			// Set ACK Timestamp	
			_TmpAlarm.AckDateTime[0] := TO_DINT(_TempTimestruct.wYear);
			_TmpAlarm.AckDateTime[1] := TO_DINT(_TempTimestruct.wMonth);
			_TmpAlarm.AckDateTime[2] := TO_DINT(_TempTimestruct.wDay);
			_TmpAlarm.AckDateTime[3] := TO_DINT(_TempTimestruct.wHour);
			_TmpAlarm.AckDateTime[4] := TO_DINT(_TempTimestruct.wMinute);
			_TmpAlarm.AckDateTime[5] := TO_DINT(_TempTimestruct.wSecond);
			_TmpAlarm.AckDateTime[6] := TO_DINT(_TempTimestruct.wMilliseconds);
			_TmpAlarm.Trigger		 := FALSE;

			// Move to History	
			_hr := THIS^.AlarmArrayHandler(NewAlarm_Ref			:= _TmpAlarm,
										   ActAlarmsCounter_Ref := THIS^.MsgInHistory,
										   MaxArrayElements		:= Tc3_PackML_V2.MaxHistoryAlarms,
										   pAlarmArray			:= ADR(_AdminTag.AlarmHistory),
										   BufferOverflow_Ref	:= _BufferOverflow);

			IF _BufferOverflow THEN
				Tc2_System.ADSLOGSTR(msgCtrlMask := Tc2_System.ADSLOG_MSGTYPE_ERROR, msgFmtStr := Tc2_Standard.CONCAT(cBaseMsg, 'MoveAlarmToHistory: %s'), strArg := 'History Buffer is full / FIFO active');
			END_IF

			IF Tc3_Module.SUCCEEDED(_hr) THEN
				// Close empty entry in source array
				Tc2_System.MEMMOVE(destAddr := ADR(pAlarmArray[_Iterator]), srcAddr := ADR(pAlarmArray[_Iterator + 1]), n := (SIZEOF(Tc3_PackML_V2.ST_Alarm) * (TO_UINT((_MaxArrayElementsInternal) - (_Iterator))))); // move Alarm 
				Tc2_System.MEMSET(destAddr := ADR(pAlarmArray[_MaxArrayElementsInternal]), fillByte := 0, n := SIZEOF(Tc3_PackML_V2.ST_Alarm));																		   // delete last entry

				// Find next empty entry index 
				FOR _Iterator2 := 0 TO (_MaxArrayElementsInternal) DO
					IF (pAlarmArray[_Iterator2].Message = '') OR (_Iterator2 = _MaxArrayElementsInternal) THEN
						IF _Iterator2 > 0 THEN
							ActAlarms_Ref := _Iterator2 - 1;
						ELSE
							ActAlarms_Ref := _Iterator2;
						END_IF

						EXIT;
					END_IF
				END_FOR
			END_IF

			EXIT;
		END_IF
	END_FOR

	MoveAlarmToHistory := S_OK;
ELSE
	// Set internal Error
	Tc2_System.ADSLOGSTR(msgCtrlMask := cMsgCtrlMask, msgFmtStr := Tc2_Standard.CONCAT(cBaseMsg, 'MoveAlarmToHistory: %s'), strArg := 'Input-reference error');
	MoveAlarmToHistory := E_FAIL;
	_InternalError	   := TRUE;
END_IF
END_METHOD

PROPERTY Name : STRING
GET
END_GET
SET
_Name := Name;
END_SET
END_PROPERTY

METHOD OnAlarmCleared : HRESULT
VAR_INPUT
	fbEvent : REFERENCE TO FB_TcEvent; // Reference to FB_Event (Callback!)
END_VAR

VAR_INST
	_idxEventReceived : INT; // Event index
END_VAR

VAR
	_hr : HRESULT; // hresult
END_VAR
// Move Alarm to History
IF fbEvent.eSeverity = TcEventSeverity.Critical THEN // Check "Critical" --> Stop reason
	_hr := MoveAlarmToHistory(MaxArrayElements := Tc3_PackML_V2.MaxStopReasons,
							  EventId		   := fbEvent.nEventId,
							  pAlarmArray	   := ADR(_AdminTag.StopReason),
							  Timestamp		   := fbEvent.nTimestamp,
							  ActAlarms_Ref	   := UnclearedStopReasons);
ELSIF fbEvent.eSeverity = TcEventSeverity.Error THEN // Check "Error" --> Alarm
	_hr := MoveAlarmToHistory(MaxArrayElements := Tc3_PackML_V2.MaxAlarms,
							  EventId		   := fbEvent.nEventId,
							  pAlarmArray	   := ADR(_AdminTag.Alarm),
							  Timestamp		   := fbEvent.nTimestamp,
							  ActAlarms_Ref	   := UnclearedAlarms);

	IF _AlarmToStopReason AND Tc3_Module.SUCCEEDED(_hr) THEN
		_hr := THIS^.ClearStopReason(pAlarmArray	  := ADR(_AdminTag.StopReason),
									 ActAlarms_Ref	  := THIS^.UnclearedStopReasons,
									 MaxArrayElements := Tc3_PackML_V2.MaxStopReasons,
									 EventId		  := fbEvent.nEventId);
	END_IF
ELSIF fbEvent.eSeverity = TcEventSeverity.Warning THEN // Check "Warning" --> Warning
	_hr := MoveAlarmToHistory(MaxArrayElements := Tc3_PackML_V2.MaxWarnings,
							  EventId		   := fbEvent.nEventId,
							  pAlarmArray	   := ADR(_AdminTag.Warning),
							  Timestamp		   := fbEvent.nTimestamp,
							  ActAlarms_Ref	   := UnclearedWarnings);

	IF _WarningToStopReason AND Tc3_Module.SUCCEEDED(_hr) THEN
		_hr := THIS^.ClearStopReason(pAlarmArray	  := ADR(_AdminTag.StopReason),
									 ActAlarms_Ref	  := THIS^.UnclearedStopReasons,
									 MaxArrayElements := Tc3_PackML_V2.MaxStopReasons,
									 EventId		  := fbEvent.nEventId);
	END_IF
END_IF

OnAlarmCleared := S_OK; // in order to receive more callbacks (Set <> S_OK in order to cancel the callbacks for this program cycle.)
END_METHOD

// Callback Method
METHOD OnAlarmConfirmed : HRESULT
VAR_INPUT
	fbEvent : REFERENCE TO FB_TcEvent; // Reference to FB_Event (Callback!)
END_VAR

VAR
	_hr : HRESULT; // hresult
END_VAR
// Move Alarm to History
IF __ISVALIDREF(fbEvent) THEN
	// Set ACK Timestamp
	IF fbEvent.eSeverity = TcEventSeverity.Critical THEN // Check "Critical" --> Stop reason
		_hr := ConfirmAlarm(MaxArrayElements := Tc3_PackML_V2.MaxStopReasons,
							EventId			 := fbEvent.nEventId,
							pAlarmArray		 := ADR(_AdminTag.StopReason),
							Timestamp		 := fbEvent.nTimestamp,
							ActAlarms_Ref	 := UnclearedStopReasons);
	ELSIF fbEvent.eSeverity = TcEventSeverity.Error THEN // Check "Error" --> Alarm
		_hr := ConfirmAlarm(MaxArrayElements := Tc3_PackML_V2.MaxAlarms,
							EventId			 := fbEvent.nEventId,
							pAlarmArray		 := ADR(_AdminTag.Alarm),
							Timestamp		 := fbEvent.nTimestamp,
							ActAlarms_Ref	 := UnclearedAlarms);
	ELSIF fbEvent.eSeverity = TcEventSeverity.Warning THEN // Check "Warning" --> Warning
		_hr := ConfirmAlarm(MaxArrayElements := Tc3_PackML_V2.MaxWarnings,
							EventId			 := fbEvent.nEventId,
							pAlarmArray		 := ADR(_AdminTag.Warning),
							Timestamp		 := fbEvent.nTimestamp,
							ActAlarms_Ref	 := UnclearedWarnings);
	END_IF

	OnAlarmConfirmed := S_OK; // in order to receive more callbacks (Set <> S_OK in order to cancel the callbacks for this program cycle.)
ELSE
	// Set internal Error
	Tc2_System.ADSLOGSTR(msgCtrlMask := cMsgCtrlMask, msgFmtStr := Tc2_Standard.CONCAT(cBaseMsg, 'OnAlarmConfirmed: %s'), strArg := 'Input-reference error');
	OnAlarmConfirmed := E_FAIL;
	_InternalError	 := TRUE;
END_IF
END_METHOD

// Callback Method
METHOD OnAlarmRaised : HRESULT
VAR_INPUT
	fbEvent : REFERENCE TO FB_TcEvent; // Reference to FB_Event (Callback!)
END_VAR

VAR
	_TempTimestruct : TIMESTRUCT; // TimeStruct for ACK Time
END_VAR
// when (new) event is triggered -> trigger within cyclic method 'execute'
THIS^.NewEvent := TRUE;

//for local event -> raise counter
CntAlarmsRaised := CntAlarmsRaised + 1;

// save eventinfo locally
THIS^.stEventInfo.Source	  := fbEvent.ipSourceInfo.sName;
THIS^.stEventInfo.eSeverity	  := fbEvent.eSeverity;
THIS^.stEventInfo.EventClass  := fbEvent.EventClass;
THIS^.stEventInfo.EventId	  := fbEvent.nEventId;
THIS^.stEventInfo.ipArguments := fbEvent.ipArguments;

// TimeZone
fbSpecificLocalTime(in := Tc2_Utilities.FILETIME64_TO_SYSTEMTIME(fbEvent.nTimestamp), tzInfo := fbTimeZone.tzInfo, out => _TempTimestruct);

// Timestamp	
THIS^.stEventInfo.TimeRaised[0] := TO_DINT(_TempTimestruct.wYear);
THIS^.stEventInfo.TimeRaised[1] := TO_DINT(_TempTimestruct.wMonth);
THIS^.stEventInfo.TimeRaised[2] := TO_DINT(_TempTimestruct.wDay);
THIS^.stEventInfo.TimeRaised[3] := TO_DINT(_TempTimestruct.wHour);
THIS^.stEventInfo.TimeRaised[4] := TO_DINT(_TempTimestruct.wMinute);
THIS^.stEventInfo.TimeRaised[5] := TO_DINT(_TempTimestruct.wSecond);
THIS^.stEventInfo.TimeRaised[6] := TO_DINT(_TempTimestruct.wMilliseconds);
Tc2_System.MEMSET(destAddr := ADR(stEventInfo.TimeCleared), fillByte := 0, n := SIZEOF(stEventInfo.TimeCleared));
Tc2_System.MEMSET(destAddr := ADR(stEventInfo.TimeConfirmed), fillByte := 0, n := SIZEOF(stEventInfo.TimeConfirmed));

//store event info globally
aEventInfoBuffer[CntAlarmsRaised] := stEventInfo;

// activate requests in event triggered method 'OnMessageSent' to get related request info
aEventInfoBuffer[CntAlarmsRaised].fbRequestEventText.Request(eventClass := aEventInfoBuffer[CntAlarmsRaised].EventClass,
															 nEventId	:= aEventInfoBuffer[CntAlarmsRaised].EventId,
															 nLangId	:= 1033,
															 ipArgs		:= aEventInfoBuffer[CntAlarmsRaised].ipArguments);

OnAlarmRaised := S_OK; // in order to receive more callbacks (Set <> S_OK in order to cancel the callbacks for this program cycle.)
END_METHOD

PROPERTY ParentResponseDefinitions : ARRAY[0..4] OF SPT_BaseTypes.E_AlarmResponse
GET
ParentResponseDefinitions := _ParentResponseDefinitions;
END_GET
SET
_ParentResponseDefinitions := ParentResponseDefinitions;
END_SET
END_PROPERTY

METHOD Reset : BOOL
//This may or may not be called depending on the component type 

//which derives FB_ComponentBase
F_ClearAllEventsInClass(PackMLEventHandlerAlarms);
Reset := TRUE;
END_METHOD

METHOD PUBLIC TimeZone : BOOL
VAR_INST
	_Step : USINT; // Step Variable
END_VAR
CASE _Step OF
	0: // Start to get local Timezone 
		fbTimeZone.bExecute := TRUE;
		IF fbTimeZone.bBusy THEN
			_Step := _Step + 1;
		END_IF

	1: // set 
		fbTimeZone.bExecute := FALSE;
		_Step				:= 0;
		TimeZone			:= TRUE;

ELSE
	Tc2_System.ADSLOGSTR(msgCtrlMask := cMsgCtrlMask, msgFmtStr := Tc2_Standard.CONCAT(cBaseMsg, 'TimeZone: %s'), strArg := 'Case Idx error');
	_InternalError := TRUE;
END_CASE

fbTimeZone(sNetID := '');
IF fbTimeZone.bError THEN
	Tc2_System.ADSLOGSTR(msgCtrlMask := cMsgCtrlMask, msgFmtStr := Tc2_Standard.CONCAT(cBaseMsg, 'fbTimeZone ErrID: %s'), strArg := TO_STRING(fbTimeZone.nErrID));
	_InternalError := TRUE;
END_IF
END_METHOD

PROPERTY WarningToStopReason : BOOL
SET
_WarningToStopReason := WarningToStopReason;
END_SET
END_PROPERTY

METHOD PRIVATE WriteAlarmTags : HRESULT;
VAR_INPUT
	Alarm_Ref	  : REFERENCE TO Tc3_PackML_V2.ST_Alarm; // Reference to ST_Alarm of an new Alarm / Warning / Stop reason
	EventInfo_Ref : REFERENCE TO ST_EventInfo;			 // Reference to ST_EventInfo
	Trigger		  : BOOL;								 // Set / Reset Trigger in PML Structure
	AlarmIndex	  : DINT;								 // Alarm index
END_VAR
IF __ISVALIDREF(Alarm_Ref) AND __ISVALIDREF(EventInfo_Ref) THEN
	Alarm_Ref.ID	   := TO_DINT(EventInfo_Ref.EventId);
	Alarm_Ref.Value	   := AlarmIndex;
	Alarm_Ref.Message  := EventInfo_Ref.EventText;
	Alarm_Ref.Category := TO_DINT(EventInfo_Ref.eSeverity); // Verbose:=0, Info:=1, Warning:=2, Error:=3, Critical:=4
	Alarm_Ref.Trigger  := Trigger;
	Alarm_Ref.DateTime := EventInfo_Ref.TimeRaised;
	WriteAlarmTags	   := S_OK;
ELSE
	// Set internal Error
	Tc2_System.ADSLOGSTR(msgCtrlMask := cMsgCtrlMask, msgFmtStr := Tc2_Standard.CONCAT(cBaseMsg, 'WriteAlarmTags: %s'), strArg := 'Input-reference error');
	WriteAlarmTags := E_FAIL;
	_InternalError := TRUE;
END_IF
END_METHOD

END_FUNCTION_BLOCK

// Project Information/F_GetCompany
// This function has been automatically generated from the project information.
{attribute 'signature_flag' := '1073741824'}
{attribute 'TcGenerated'}
{attribute 'no-analysis'}
FUNCTION F_GetCompany : WSTRING
VAR_INPUT
	
END_VAR

F_GetCompany := "Beckhoff Automation LLC";

END_FUNCTION

// Project Information/F_GetTitle
// This function has been automatically generated from the project information.
{attribute 'signature_flag' := '1073741824'}
{attribute 'TcGenerated'}
{attribute 'no-analysis'}
FUNCTION F_GetTitle : WSTRING
VAR_INPUT
	
END_VAR

F_GetTitle := "SPT Components";

END_FUNCTION

// Project Information/F_GetVersion
// This function has been automatically generated from the project information.
{attribute 'signature_flag' := '1073741824'}
{attribute 'TcGenerated'}
{attribute 'no-analysis'}
FUNCTION F_GetVersion : ST_LibVersion
VAR_INPUT
	
END_VAR

F_GetVersion.iMajor := 3;
F_GetVersion.iMinor := 2;
F_GetVersion.iBuild := 6;
F_GetVersion.iRevision := 0;
F_GetVersion.sVersion := '3.2.6';
F_GetVersion.nFlags := 1;

END_FUNCTION

// Sensors/FB_DigitalSensor
FUNCTION_BLOCK FB_DigitalSensor EXTENDS FB_ComponentBase IMPLEMENTS I_DigitalSensorBase
VAR
	HardwareInput AT %I*		: BOOL;			  //Hardware input bit from the hysical sensor
	_DebounceMode				: E_DebounceMode; //Defines the debounce model that will filter the sensor's output to the program
	_DebounceTime				: TIME;			  //Time input parameter for use in Debounce functionality
	_Inverted					: BOOL;			  //Defines the output polarity of the sensor - a "TRUE" value will result in the signal of the sensor being inverted
	_SimulationInput			: BOOL;			  //Provides configuration input to the simulation functionality
	_SimulationTimebase			: UDINT;
	_SimulationMode				: E_SensorSimulationMode; //Defines the mode of operation for the simulation functionality of this component
	_TimeActive					: TIME;					  //Tracks the amount of time that the sensor has been in an active state
	_TimeInactive				: TIME;					  //Tracks the amount of time that the sensor has been in an inactive state
	_Active						: BOOL;
	TON_ActiveTimer				: Tc2_Standard.TON; //Tracks the amount of time that the sensor has been in an active state
	TON_InactiveTimer			: Tc2_Standard.TON; //Tracks the amount of time that the sensor has been in an inactive state
	TON_DebounceTimer			: Tc2_Standard.TON; //Utilized in the debounce implementation
	TP_DebounceTimer			: Tc2_Standard.TP;	//Utilized in the debounce implementation
	DigitalSensor_HMI			: ST_DigitalSensor_HMI;
	SimulationPulse1_TP			: Tc2_Standard.TP; //Pulse Timer for simulated sensor pulse generation
	SimulationPulse2_TP			: Tc2_Standard.TP; //Pulse Timer for simulated sensor pulse generation
	HMICommand_DigitalSensor_RT : R_TRIG;
END_VAR

METHOD PUBLIC CyclicLogic
VAR_INPUT
END_VAR
SUPER^.CyclicLogic();
IF _Simulate THEN
	CASE _SimulationMode OF
		E_SensorSimulationMode.InputDriven:
			_Active := _SimulationInput;

		E_SensorSimulationMode.Periodic:
			SimulationPulse1_TP(IN := NOT SimulationPulse2_TP.Q, PT := UDINT_TO_TIME(_SimulationTimebase));
			SimulationPulse2_TP(IN := NOT SimulationPulse1_TP.Q, PT := UDINT_TO_TIME(_SimulationTimebase));
			_Active := SimulationPulse2_TP.Q;
	END_CASE
ELSE
	_Active := ProcessInput(Input := HardwareInput);
END_IF
END_METHOD

PROPERTY Active : BOOL
GET
Active := _Active;
END_GET
END_PROPERTY

PROPERTY DebounceMode : E_DebounceMode
GET
DebounceMode := _DebounceMode;
END_GET
SET
_DebounceMode := DebounceMode;
END_SET
END_PROPERTY

PROPERTY DebounceTime : TIME
GET
DebounceTime := _DebounceTime;
END_GET
SET
_DebounceTime := DebounceTime;
END_SET
END_PROPERTY

PROPERTY Inverted : BOOL
GET
Inverted := _Inverted;
END_GET
SET
_Inverted := Inverted;
END_SET
END_PROPERTY

PROPERTY SimulationInput : BOOL
GET
SimulationInput := _SimulationInput;
END_GET
SET
_SimulationInput := SimulationInput;
END_SET
END_PROPERTY

PROPERTY SimulationMode : E_SensorSimulationMode
GET
SimulationMode := _SimulationMode;
END_GET
SET
_SimulationMode := SimulationMode;
END_SET
END_PROPERTY

PROPERTY SimulationTimeBase : UDINT
GET
SimulationTimeBase := _SimulationTimebase;
END_GET
SET
_SimulationTimeBase := SimulationTimebase;
END_SET
END_PROPERTY

PROPERTY TimeActive : TIME
GET
TimeActive := _TimeActive;
END_GET
END_PROPERTY

PROPERTY TimeInactive : TIME
GET
TimeInactive := _TimeInactive;
END_GET
END_PROPERTY

METHOD PROTECTED HMICommunication
//Extend this method in extended FBs to communicate specific implementation data
SUPER^.HMICommunication();

//Process HMI requests

//Replace 'FALSE' below with further momentary commands (myCommand XOR myOtherCommand XOR...)
HMICommand_DigitalSensor_RT(CLK := (ComponentBase_HMI.Status.HMIControlAvailable AND NOT HMICommandActive_Base) AND (FALSE));

//Signal to FB_ComponentBase that a command is active
HMICommandActive_Descendant := ComponentBase_HMI.Status.HMIControlAvailable AND (DigitalSensor_HMI.Config.DebounceMode <> _DebounceMode OR DigitalSensor_HMI.Config.DebounceTime <> _DebounceTime OR DigitalSensor_HMI.Config.Inverted <> _Inverted OR DigitalSensor_HMI.Config.SimulationMode <> _SimulationMode OR DigitalSensor_HMI.Config.SimulationTimebase <> _SimulationTimebase);

//Process HMI requests
IF HMICommand_DigitalSensor_RT.Q THEN //If a request has been issued by the HMI, and a previous request has not just finished being processed

	//	IF AxisBaseHMI.Command.xxx THEN

	//		Enabled := TRUE;

	//	END_IF
END_IF

IF ComponentBase_HMI.Status.HMIControlAvailable AND NOT HMICommand_DigitalSensor_RT.Q THEN
	IF DigitalSensor_HMI.Config.DebounceMode <> _DebounceMode THEN
		DebounceMode := DigitalSensor_HMI.Config.DebounceMode;
	END_IF

	IF DigitalSensor_HMI.Config.DebounceTime <> _DebounceTime THEN
		DebounceTime := DigitalSensor_HMI.Config.DebounceTime;
	END_IF

	IF DigitalSensor_HMI.Config.Inverted <> _Inverted THEN
		Inverted := DigitalSensor_HMI.Config.Inverted;
	END_IF

	IF DigitalSensor_HMI.Config.SimulationMode <> _SimulationMode THEN
		SimulationMode := DigitalSensor_HMI.Config.SimulationMode;
	END_IF

	IF DigitalSensor_HMI.Config.SimulationTimebase <> _SimulationTimebase THEN
		SimulationTimeBase := DigitalSensor_HMI.Config.SimulationTimebase;
	END_IF
END_IF

//Update HMI status info
DigitalSensor_HMI.Status.Active				:= _Active;
DigitalSensor_HMI.Status.TimeActive			:= TIME_TO_LREAL(_TimeActive) / 1000.0;
DigitalSensor_HMI.Status.TimeInactive		:= TIME_TO_LREAL(_TimeInactive) / 1000.0;
DigitalSensor_HMI.Config.DebounceMode		:= DebounceMode;
DigitalSensor_HMI.Config.DebounceTime		:= DebounceTime;
DigitalSensor_HMI.Config.Inverted			:= Inverted;
DigitalSensor_HMI.Config.SimulationMode		:= SimulationMode;
DigitalSensor_HMI.Config.SimulationTimebase := SimulationTimeBase;
END_METHOD

METHOD PROTECTED Monitoring
SUPER^.Monitoring();

//If flicker counters or other diagnostic systems are desired, their implementation could be here

//Any warnings, errors, or other desired messages would also be generated here

//T#71582M47S295MS is the upper bound of the TIME type, meaning these timers will continue to increase ET for as long as possible
TON_ActiveTimer(IN := _Active, PT := T#71582M47S295MS, ET => _TimeActive);
TON_InactiveTimer(IN := NOT _Active, PT := T#71582M47S295MS, ET => _TimeInactive);
_Busy  := FALSE;
_Error := FALSE;
END_METHOD

METHOD PRIVATE ProcessInput : BOOL
VAR_INPUT
	Input : BOOL;
END_VAR

VAR
	DebouncedInput : BOOL;
END_VAR

VAR_INST
	LastDebouncedInput : BOOL;
	MovingAverage	   : DINT;
END_VAR
CASE DebounceMode OF
	E_DebounceMode.RawInput: //Passes raw input through
		DebouncedInput := Input;

	E_DebounceMode.SimpleFlickerFilter:											 //Requires the raw input to be a consistent value for a set time period before output changes
		TON_DebounceTimer(IN := (Input <> DebouncedInput), PT := _DebounceTime); //runs the timer whenever a differing input is detected
		IF TON_DebounceTimer.Q THEN
			DebouncedInput := Input; //once the raw input has been different for the specified debounce time, the processed input is updated
		END_IF

	E_DebounceMode.EdgeDetectFilter:								   //Updates the processed value immediately on a change from steady state, but mutes any sensor flickers for the specified time immediately following the change
		IF (Input <> DebouncedInput) AND (NOT TP_DebounceTimer.Q) THEN //A differing raw input must be detected outside of the mute window created by the pulse timer
			DebouncedInput := Input;
		END_IF

		TP_DebounceTimer(IN := (DebouncedInput <> LastDebouncedInput), PT := _DebounceTime); //"Q" will be TRUE for tDebounce time after the bProcessedSensorInput value is changed
	E_DebounceMode.MovingAverage:															 //Uses a "moving average"-like calculation to compensate for extremely inconsistent signals - prevents poorly timed flickers from causing disproportionate results
		TON_DebounceTimer(IN := NOT TON_DebounceTimer.Q, PT := T#5MS);						 //Provides a 1ms "polling" trigger
		IF TON_DebounceTimer.Q THEN															 //TRUE once every millisecond
			IF Input THEN																	 //If raw input is currently active at the time of polling
				IF MovingAverage < TIME_TO_DINT(_DebounceTime) THEN							 //If the moving average has not reached its "weight limit" as set by debounce time
					MovingAverage := MovingAverage + 5;										 //Add 1 to the average
				END_IF
			ELSE													 //If raw input is currently inactive at the time of polling
				IF MovingAverage > -TIME_TO_DINT(_DebounceTime) THEN //If the moving average has not reached its "weight limit" as set by debounce time
					MovingAverage := MovingAverage - 5;				 //Subtract 1 from the average
				END_IF
			END_IF
		END_IF

		IF MovingAverage >= 0 THEN
			DebouncedInput := TRUE;
		ELSE
			DebouncedInput := FALSE;
		END_IF
END_CASE

LastDebouncedInput := DebouncedInput; //Update "Last value"
IF _Inverted THEN					  //If signal inversion is requested, invert the signal
	DebouncedInput := NOT DebouncedInput;
END_IF

ProcessInput := DebouncedInput;
END_METHOD

END_FUNCTION_BLOCK

// Sensors/I_DigitalSensorBase
INTERFACE I_DigitalSensorBase

PROPERTY Active : BOOL
GET
END_GET
END_PROPERTY

PROPERTY DebounceMode : E_DebounceMode
GET
END_GET
SET
END_SET
END_PROPERTY

PROPERTY DebounceTime : TIME
GET
END_GET
SET
END_SET
END_PROPERTY

PROPERTY Inverted : BOOL //"High" signal from the sensor will be interpreted as an "inactive" reading when this parameter is TRUE
GET
END_GET
SET
END_SET
END_PROPERTY

PROPERTY SimulationInput : BOOL
GET
END_GET
SET
END_SET
END_PROPERTY

PROPERTY SimulationMode : E_SensorSimulationMode
GET
END_GET
SET
END_SET
END_PROPERTY

PROPERTY TimeActive : TIME
GET
END_GET
END_PROPERTY

PROPERTY TimeInactive : TIME
GET
END_GET
END_PROPERTY

END_INTERFACE

// Solenoids/SolenoidBankBase/FB_SolenoidBankBase
FUNCTION_BLOCK ABSTRACT FB_SolenoidBankBase EXTENDS FB_ComponentBase
VAR
	// Configuration
	Configuration : ARRAY[1..Parameters_Cylinder.MAX_NUMBER_OF_SOLENOIDS] OF ST_SolenoidBankConfig;

	//Counted number of solenoids
	NumberOfSolenoids : UINT;

	//Alarms
	SolenoidBankAlarms : ARRAY[1..SolenoidBankBaseAlarmsCount] OF FB_TcAlarm;
END_VAR

VAR CONSTANT
	SolenoidBankBaseAlarmsCount : UINT := 2;
END_VAR

METHOD PUBLIC AddSolenoid : UINT
VAR_INPUT
	ipCylinder	 : I_Solenoid;
	Number		 : UINT; //This is the number in the IO tree.
	SolenoidType : E_SolenoidType;
END_VAR
IF CheckNumber(Number) AND ipCylinder <> 0 THEN
	NumberOfSolenoids									  := NumberOfSolenoids + 1;
	Configuration[NumberOfSolenoids].ipSolenoid			  := ipCylinder;
	Configuration[NumberOfSolenoids].SolenoidType		  := SolenoidType;
	Configuration[NumberOfSolenoids].SolenoidOutputNumber := Number;
END_IF
END_METHOD

METHOD PRIVATE CheckNumber : BOOL
VAR_INPUT
	Number : UINT;
END_VAR
CheckNumber := TRUE;
IF Number < 1 AND Number > Parameters_Cylinder.MAX_NUMBER_OF_SOLENOIDS THEN
	IF NOT SolenoidBankAlarms[E_CylinderBankAlarms.CylinderNumberOutOfRange].bRaised THEN
		SolenoidBankAlarms[E_CylinderBankAlarms.CylinderNumberOutOfRange].Raise(0);
	END_IF

	CheckNumber := FALSE;
END_IF
END_METHOD

METHOD PROTECTED CreateEvents
SUPER^.CreateEvents();
F_CreateAllEventsInClass(Alarms		:= SolenoidBankAlarms,
						 ClassSize	:= SIZEOF(TC_EVENTS.CylinderBankAlarms),
						 pInitEvent := ADR(TC_EVENTS.CylinderBankAlarms.InitReferenceEvent),
						 Prefix		:= Name);
END_METHOD

//! @summary This method serves as the entry point for all underlying FB logic
METHOD PUBLIC CyclicLogic
//! @description This method should be called cyclically by descendant function blocks by invoking <c>SUPER^.CyclicLogic()</c>.  Alternatively, the contents of this method could be reimplemented entirely in which case a call to this method would not be necessary.
VAR
	x : UINT;
END_VAR
//Loop through all solenoids that are added.
FOR x := 1 TO NumberOfSolenoids DO
	MapIO(x);
END_FOR
END_METHOD

//! @summary Basic component initialization logic
METHOD PROTECTED Initialize : BOOL;
//! @description This method is called by <c>CyclicLogic()</c> as required
VAR
	x : UINT;
END_VAR
NumberOfSolenoids := 0;
Initialize		  := TRUE;
END_METHOD

METHOD ABSTRACT MapIO
VAR_INPUT
	x : UINT;
END_VAR
END_METHOD

//! Provides basic error detection and event handling for this component
METHOD PROTECTED Monitoring

(*! @descriptionThis method is called cyclically by <c>CyclicLogic()</c>*)
SUPER^.Monitoring();
_CurrentAlarmSeverity := F_GetMaxSeverityRaised(Alarms := SolenoidBankAlarms, CurrentSeverity := CurrentAlarmSeverity);
END_METHOD

//! @summary Clears error flags and error IDs for this component
METHOD PUBLIC Reset : BOOL
SUPER^.Reset();
IF SolenoidBankAlarms[E_CylinderBankAlarms.CylinderNumberOutOfRange].bRaised THEN
	SolenoidBankAlarms[E_CylinderBankAlarms.CylinderNumberOutOfRange].Clear(0, 0);
END_IF
END_METHOD

END_FUNCTION_BLOCK

// Solenoids/I_Solenoid
INTERFACE I_Solenoid

METHOD Extend
VAR_INPUT
END_VAR
END_METHOD

PROPERTY Extended : BOOL
GET
END_GET
END_PROPERTY

PROPERTY ExtendOutput : BOOL
GET
END_GET
END_PROPERTY

PROPERTY ExtendTime : LREAL
GET
END_GET
SET
END_SET
END_PROPERTY

METHOD Retract
VAR_INPUT
END_VAR
END_METHOD

PROPERTY Retracted : BOOL
GET
END_GET
END_PROPERTY

PROPERTY RetractOutput : BOOL
GET
END_GET
END_PROPERTY

PROPERTY RetractTime : LREAL
GET
END_GET
SET
END_SET
END_PROPERTY

END_INTERFACE

// Solenoids/FB_DoubleSolenoid
FUNCTION_BLOCK FB_DoubleSolenoid EXTENDS FB_SingleSolenoid
VAR
	_RetractOutput AT %Q* : BOOL;
END_VAR

METHOD PROTECTED HardwareInit
//Update the status based on the IO 
IF _ExtendOutput AND NOT _RetractOutput THEN
	_Extended  := TRUE;
	_Retracted := FALSE;
ELSIF NOT _ExtendOutput AND _RetractOutput THEN
	_Extended  := FALSE;
	_Retracted := TRUE;
ELSE // By Default, set RetractOuptupt if neither is set or if both are set.
	_ExtendOutput  := FALSE;
	_RetractOutput := TRUE;
	_Extended	   := FALSE;
	_Retracted	   := TRUE;
END_IF
END_METHOD

METHOD PROTECTED HardwareUpdate
//One shot the requests
Extend_RTRIG(CLK := _ExtendRequest);
Retract_RTRIG(CLK := _RetractRequest);

//Handle Extend
IF Extend_RTRIG.Q THEN
	_ExtendOutput	:= TRUE;
	_RetractOutput	:= FALSE;
	_Extending		:= TRUE;
	_Retracting		:= FALSE;
	_Retracted		:= FALSE;
	_RetractRequest := FALSE;
END_IF

//Handle Retract
IF Retract_RTRIG.Q THEN
	_ExtendOutput  := FALSE;
	_RetractOutput := TRUE;
	_Extending	   := FALSE;
	_Retracting	   := TRUE;
	_Extended	   := FALSE;
	_ExtendRequest := FALSE;
END_IF

//Always Simulate Feedback here with no feedback inputs
Feedback();
END_METHOD

PROPERTY RetractOutput : BOOL
GET
RetractOutput := _RetractOutput;
END_GET
END_PROPERTY

END_FUNCTION_BLOCK

// Solenoids/FB_SingleSolenoid
(*	This FB is used for a single output solenoid 
	It uses the times to say when Extended/Retracted  	
	It starts assuming retracted and the output off.
*)
FUNCTION_BLOCK FB_SingleSolenoid EXTENDS FB_ComponentBase IMPLEMENTS I_Solenoid
VAR
	//Output
	_ExtendOutput AT %Q* : BOOL;

	// Internal variables
	_ExtendRequest	: BOOL;
	_RetractRequest : BOOL;
	_Extended		: BOOL;
	_Retracted		: BOOL;
	_Extending		: BOOL;
	_Retracting		: BOOL;
	_ExtendTime		: LREAL := 1000; // Default time 1s
	_RetractTime	: LREAL := 1000; // Default time 1s

	// Timer for Extend/Retract
	Extend_TON	  : TON;
	Retract_TON	  : TON;
	Extend_RTRIG  : R_TRIG;
	Retract_RTRIG : R_TRIG;

	//HMI 
	SolenoidHMI : ST_Cylinder_HMI;

	//Alarms
	SolenoidAlarms : ARRAY[1..SolenoidAlarmsCount] OF FB_TcAlarm;
END_VAR

VAR CONSTANT
	SolenoidAlarmsCount : UINT := 4;
END_VAR

METHOD PROTECTED CreateEvents
SUPER^.CreateEvents();
F_CreateAllEventsInClass(Alarms		:= SolenoidAlarms,
						 ClassSize	:= SIZEOF(TC_EVENTS.CylinderAlarms),
						 pInitEvent := ADR(TC_EVENTS.CylinderAlarms.InitReferenceEvent),
						 Prefix		:= Name);
END_METHOD

METHOD PROTECTED HMICommunication
VAR_INPUT
END_VAR
SUPER^.HMICommunication();

//Handle the requests to extend and retract
IF ComponentBase_HMI.Status.HMIControlAvailable THEN
	IF SolenoidHMI.Command.Extend THEN
		Extend();
	ELSIF SolenoidHMI.Command.Retract THEN
		Retract();
	END_IF

	IF NOT F_CompareLREAL(SolenoidHMI.Command.ExtendTime, _ExtendTime, 0.01) THEN
		_ExtendTime := SolenoidHMI.Command.ExtendTime;
	END_IF

	IF NOT F_CompareLREAL(SolenoidHMI.Command.RetractTime, _RetractTime, 0.01) THEN
		_RetractTime := SolenoidHMI.Command.RetractTime;
	END_IF
END_IF

//Update HMI status info
SolenoidHMI.Status.Extended	   := _Extended;
SolenoidHMI.Status.Extending   := _Extending;
SolenoidHMI.Status.Retracted   := _Retracted;
SolenoidHMI.Status.Retracting  := _Retracting;
SolenoidHMI.Config.ExtendTime  := _ExtendTime;
SolenoidHMI.Config.RetractTime := _RetractTime;
END_METHOD

METHOD PROTECTED Monitoring
VAR_INPUT
END_VAR
SUPER^.Monitoring();

//Update output bits
_Busy				  := _Extending OR _Retracting;
_CurrentAlarmSeverity := F_GetMaxSeverityRaised(Alarms := SolenoidAlarms, CurrentSeverity := CurrentAlarmSeverity);
_Error				  := _CurrentAlarmSeverity >= TcEventSeverity.Error;
END_METHOD

METHOD CyclicLogic
VAR
	myErrorID : UDINT;
END_VAR
HardwareUpdate();
SUPER^.CyclicLogic();

//New code
myErrorID := THIS^.ErrorID;
END_METHOD

METHOD Extend
_ExtendRequest	:= TRUE;
_RetractRequest := FALSE;
END_METHOD

PROPERTY Extended : BOOL
GET
Extended := _Extended;
END_GET
END_PROPERTY

PROPERTY ExtendOutput : BOOL
GET
ExtendOutput := _ExtendOutput;
END_GET
END_PROPERTY

PROPERTY ExtendTime : LREAL
GET
ExtendTime := _ExtendTime;
END_GET
SET
_ExtendTime					   := ExtendTime;
SolenoidHMI.Command.ExtendTime := ExtendTime;
END_SET
END_PROPERTY

METHOD Retract
_ExtendRequest	:= FALSE;
_RetractRequest := TRUE;
END_METHOD

PROPERTY Retracted : BOOL
GET
Retracted := _Retracted;
END_GET
END_PROPERTY

PROPERTY RetractOutput : BOOL
GET
RetractOutput := FALSE;
END_GET
END_PROPERTY

PROPERTY RetractTime : LREAL
GET
RetractTime := _RetractTime;
END_GET
SET
_RetractTime					:= RetractTime;
SolenoidHMI.Command.RetractTime := RetractTime;
END_SET
END_PROPERTY

METHOD PROTECTED Feedback
VAR_INPUT
END_VAR
//Handle the time to Extend/Retract
Extend_TON(IN := _Extending, PT := LREAL_TO_TIME(_ExtendTime));
Retract_TON(IN := _Retracting, PT := LREAL_TO_TIME(_RetractTime));
IF Extend_TON.Q THEN
	_Extended  := TRUE;
	_Extending := FALSE;
END_IF

IF Retract_TON.Q THEN
	_Retracted	:= TRUE;
	_Retracting := FALSE;
END_IF
END_METHOD

METHOD PROTECTED HardwareInit
IF _ExtendOutput THEN
	_Extended  := TRUE;
	_Retracted := FALSE;
ELSE
	_Extended  := FALSE;
	_Retracted := TRUE;
END_IF
END_METHOD

METHOD PROTECTED HardwareUpdate
VAR_INPUT
END_VAR
//One shot the requests
Extend_RTRIG(CLK := _ExtendRequest);
Retract_RTRIG(CLK := _RetractRequest);

//Handle Extend
IF Extend_RTRIG.Q THEN
	_ExtendOutput	:= TRUE;
	_Extending		:= TRUE;
	_Retracting		:= FALSE;
	_Retracted		:= FALSE;
	_RetractRequest := FALSE;
END_IF

//Handle Retract
IF Retract_RTRIG.Q THEN
	_ExtendOutput  := FALSE;
	_Extending	   := FALSE;
	_Retracting	   := TRUE;
	_Extended	   := FALSE;
	_ExtendRequest := FALSE;
END_IF

//Call the feedback 
Feedback();
END_METHOD

//! @summary Basic component initialization logic
METHOD PROTECTED Initialize : BOOL;

//! @description This method is called by <c>CyclicLogic()</c> as required
//Set the cylinder to retracted
_Extending		:= FALSE;
_ExtendRequest	:= FALSE;
_Retracting		:= FALSE;
_RetractRequest := FALSE;

//Set the HMI time to the currnt time.
SolenoidHMI.Command.ExtendTime	:= _ExtendTime;
SolenoidHMI.Command.RetractTime := _RetractTime;

//Call base class Initialize
Initialize := SUPER^.Initialize();

// Call the HardwareInit
HardwareInit();
END_METHOD

//! @summary Clears error flags and error IDs for this component
METHOD PUBLIC Reset : BOOL
SUPER^.Reset();
F_ClearAllEventsInClass(Alarms := SolenoidAlarms);
Reset := TRUE;
END_METHOD

END_FUNCTION_BLOCK

// Solenoids/FB_DoubleSolenoidFeedback
FUNCTION_BLOCK FB_DoubleSolenoidFeedback EXTENDS FB_DoubleSolenoid
VAR
	ExtendedSensor	AT %I* : BOOL;
	RetractedSensor AT %I* : BOOL;
END_VAR

PROPERTY ExtendedInput : BOOL
SET
ExtendedSensor := ExtendedInput;
END_SET
END_PROPERTY

METHOD PROTECTED Feedback
IF NOT _Simulate THEN
	_Extended  := ExtendedSensor;
	_Retracted := RetractedSensor;
	Extend_TON(IN := _Extending, PT := LREAL_TO_TIME(_ExtendTime));
	Retract_TON(IN := _Retracting, PT := LREAL_TO_TIME(_RetractTime));
	IF Extend_TON.Q AND NOT ExtendedSensor THEN
		IF NOT SolenoidAlarms[E_CylinderAlarms.ExtendTimeout].bRaised THEN
			SolenoidAlarms[E_CylinderAlarms.ExtendTimeout].Raise(0);
			_ExtendRequest := FALSE;
			_Extending	   := FALSE;
		END_IF
	ELSIF _Extending AND ExtendedSensor THEN
		_Extended  := TRUE;
		_Extending := FALSE;
	END_IF

	IF Retract_TON.Q AND NOT RetractedSensor THEN
		IF NOT SolenoidAlarms[E_CylinderAlarms.RetractTimeout].bRaised THEN
			SolenoidAlarms[E_CylinderAlarms.RetractTimeout].Raise(0);
			_RetractRequest := FALSE;
			_Retracting		:= FALSE;
		END_IF
	ELSIF _Retracting AND RetractedSensor THEN
		_Retracted	:= TRUE;
		_Retracting := FALSE;
	END_IF
ELSE
	SUPER^.Feedback();
END_IF

//Monitor Inputs in case both on at the same time
IF ExtendedSensor AND RetractedSensor AND NOT SolenoidAlarms[E_CylinderAlarms.ExtendedAndRetracted].bRaised THEN
	SolenoidAlarms[E_CylinderAlarms.ExtendedAndRetracted].Raise(0);
ELSIF (ExtendedSensor XOR RetractedSensor) AND SolenoidAlarms[E_CylinderAlarms.ExtendedAndRetracted].bRaised THEN
	SolenoidAlarms[E_CylinderAlarms.ExtendedAndRetracted].Clear(0, 0);
END_IF
END_METHOD

METHOD PROTECTED HardwareInit
IF ExtendedSensor AND NOT RetractedSensor THEN
	_Extended  := TRUE;
	_Retracted := FALSE;
ELSIF NOT ExtendedSensor AND RetractedSensor THEN
	_Extended  := FALSE;
	_Retracted := TRUE;
ELSE // With Neither on, then this means that it is not either or maybe no air
	_Extended  := FALSE;
	_Retracted := FALSE;
END_IF
END_METHOD

PROPERTY RetractedInput : BOOL
SET
RetractedSensor := RetractedInput;
END_SET
END_PROPERTY

END_FUNCTION_BLOCK

// Solenoids/FB_SingleSolenoidFeedback
FUNCTION_BLOCK FB_SingleSolenoidFeedback EXTENDS FB_SingleSolenoid
VAR
	ExtendedSensor	AT %I* : BOOL;
	RetractedSensor AT %I* : BOOL;
END_VAR

PROPERTY ExtendedInput : BOOL
SET
ExtendedSensor := ExtendedInput;
END_SET
END_PROPERTY

METHOD PROTECTED Feedback
IF NOT _Simulate THEN
	_Extended  := ExtendedSensor;
	_Retracted := RetractedSensor;
	Extend_TON(IN := _Extending, PT := LREAL_TO_TIME(_ExtendTime));
	Retract_TON(IN := _Retracting, PT := LREAL_TO_TIME(_RetractTime));
	IF Extend_TON.Q AND NOT ExtendedSensor THEN
		IF NOT SolenoidAlarms[E_CylinderAlarms.ExtendTimeout].bRaised THEN
			SolenoidAlarms[E_CylinderAlarms.ExtendTimeout].Raise(0);
			_ExtendRequest := FALSE;
			_Extending	   := FALSE;
		END_IF
	ELSIF _Extending AND ExtendedSensor THEN
		_Extended  := TRUE;
		_Extending := FALSE;
	END_IF

	IF Retract_TON.Q AND NOT RetractedSensor THEN
		IF NOT SolenoidAlarms[E_CylinderAlarms.RetractTimeout].bRaised THEN
			SolenoidAlarms[E_CylinderAlarms.RetractTimeout].Raise(0);
			_RetractRequest := FALSE;
			_Retracting		:= FALSE;
		END_IF
	ELSIF _Retracting AND RetractedSensor THEN
		_Retracted	:= TRUE;
		_Retracting := FALSE;
	END_IF
ELSE
	SUPER^.Feedback(); //Call the feedback that usese timers for feedback
END_IF

//Monitor Inputs in case both on at the same time
IF ExtendedSensor AND RetractedSensor AND NOT SolenoidAlarms[E_CylinderAlarms.ExtendedAndRetracted].bRaised THEN
	SolenoidAlarms[E_CylinderAlarms.ExtendedAndRetracted].Raise(0);
ELSIF (ExtendedSensor XOR RetractedSensor) AND SolenoidAlarms[E_CylinderAlarms.ExtendedAndRetracted].bRaised THEN
	SolenoidAlarms[E_CylinderAlarms.ExtendedAndRetracted].Clear(0, 0);
END_IF
END_METHOD

METHOD PROTECTED HardwareInit
IF ExtendedSensor AND NOT RetractedSensor THEN
	_Extended  := TRUE;
	_Retracted := FALSE;
ELSIF NOT ExtendedSensor AND RetractedSensor THEN
	_Extended  := FALSE;
	_Retracted := TRUE;
ELSE // With Neither on, then this means that it is not either or maybe no air
	_Extended  := FALSE;
	_Retracted := FALSE;
END_IF
END_METHOD

PROPERTY RetractedInput : BOOL
SET
RetractedSensor := RetractedInput;
END_SET
END_PROPERTY

END_FUNCTION_BLOCK

// Testing/Axis/FB_ComponentBasicAxis_Test
FUNCTION_BLOCK FB_ComponentBasicAxis_Test EXTENDS TCUnit.FB_TestSuite
VAR
	TestFBInit					: FB_Component_BasicAxis;
	TestFBNameSetProperty		: FB_Component_BasicAxis;
	TestFBSimulationSetProperty : FB_Component_BasicAxis;
	TestFBSimulationSetHMI		: FB_Component_BasicAxis;
	TestFBSimulationCheckAlarm	: FB_Component_BasicAxis;
	TestFBBusy					: FB_Component_BasicAxis;
	TestFBAllowHMI				: FB_Component_BasicAxis;
	TestFBBlockHMI				: FB_Component_BasicAxis;

	//Axis integration test - this should be tested in the NCAxis library. (Enable, Disable, etc....)

	//Alarm Testing - 17 Alarms with FB_ComponentBasicAxis

	///TestFBAlarm1  FB_Component_BasicAxis; // InitReference (Not an actual alarm)
	TestFBAlarm2 : FB_Component_BasicAxis; // MC_Power
	TestFBAlarm3 : FB_Component_BasicAxis; // MC_Reset
	TestFBAlarm4 : FB_Component_BasicAxis; // MC_Halt

	///TestFBAlarm5 FB_Component_BasicAxis; // MC_Stop // Not Implemented
	TestFBAlarm6  : FB_Component_BasicAxis; // MC_Home
	TestFBAlarm7  : FB_Component_BasicAxis; // MC_Jog
	TestFBAlarm8  : FB_Component_BasicAxis; // MC_MoveAbsolute
	TestFBAlarm9  : FB_Component_BasicAxis; // MC_MoveRelative
	TestFBAlarm10 : FB_Component_BasicAxis; // MC_MoveVelocity
	TestFBAlarm11 : FB_Component_BasicAxis; // MC_MoveModulo
	TestFBAlarm12 : FB_Component_BasicAxis; // MC_ReadParameter
	TestFBAlarm13 : FB_Component_BasicAxis; // MC_WriteParameter
	TestFBAlarm14 : FB_Component_BasicAxis; // MC_WriteBOOLParameter
	TestFBAlarm15 : FB_Component_BasicAxis; // Command While Inhibited

	///TestFBAlarm16 FB_Component_BasicAxis; // Axis Error (Not Sure how to get Axis error with virtual axis)

	///TestFBAlarm17 FB_Component_BasicAxis; // Drive Error (Cannot Get Drive Error without drive)
END_VAR

Init();
NameSetProperty();
SimulationSetProperty();
SimulationSetHMI();
SimulationCheckAlarm();
Busy();
AllowHMI();
BlockHMI();

//Tests for Alarms
MCPowerAlarm();
MCResetAlarm();
MCHaltAlarm();
MCHomeAlarm();
MCJogAlarm();
MCMoveAbsoluteAlarm();
MCMoveRelativeAlarm();
MCMoveVelocity();
MCMoveModulo();
McReadAxisParametersAlarm();
McWriteAxisParameterAlarm();
McWriteAxisBoolParameterAlarm();
CommandInhibited();

METHOD AllowHMI
VAR_INST
	State		   : INT;
	ActualResult   : BOOL;
	ExpectedResult : BOOL := TRUE;
END_VAR
IF TEST_ORDERED('BasicAxisAllowHMI') THEN
	CASE State OF
		0:
			State := State + 10;

		10:
			IF TestFBAllowHMI.InitComplete AND NOT TestFBAllowHMI.Busy THEN
				TestFBAllowHMI.AllowHMIControl();
				State := State + 10;
			END_IF

		20:
			ActualResult := TestFBAllowHMI.ComponentBase_HMI.Status.HMIControlAvailable;
			AssertEquals_BOOL(Expected := ExpectedResult, Actual := ActualResult, Message := 'Function Block read allow HMI Control in HMI Tag not true');
			TEST_FINISHED();
			State := State + 10;
	END_CASE

	//Call to FB Cyclic Logic
	TestFBAllowHMI.CyclicLogic();
END_IF
END_METHOD

METHOD BlockHMI
VAR_INST
	State		   : INT;
	ActualResult   : BOOL;
	ExpectedResult : BOOL := FALSE;
END_VAR
IF TEST_ORDERED('BasicAxisBlockHMI') THEN
	CASE State OF
		0:
			State := State + 10;

		10:
			IF TestFBBlockHMI.InitComplete AND NOT TestFBBlockHMI.Busy THEN
				TestFBBlockHMI.AllowHMIControl();
				State := State + 10;
			END_IF

		20:
			IF TestFBBlockHMI.ComponentBase_HMI.Status.HMIControlAvailable THEN
				TestFBBlockHMI.BlockHMIControl();
				State := State + 10;
			END_IF

		30:
			ActualResult := TestFBBlockHMI.ComponentBase_HMI.Status.HMIControlAvailable;
			AssertEquals_BOOL(Expected := ExpectedResult, Actual := ActualResult, Message := 'Function Block read Block HMI Control in HMI Tag not false');
			TEST_FINISHED();
			State := State + 10;
	END_CASE

	//Call to FB Cyclic Logic
	TestFBBlockHMI.CyclicLogic();
END_IF
END_METHOD

METHOD Busy
VAR_INST
	State		   : INT;
	ActualResult   : BOOL;
	ExpectedResult : BOOL := TRUE;
	Timeout		   : TON;
END_VAR
IF TEST_ORDERED('BasicAxisBusy') THEN
	CASE State OF
		0:
			State := State + 10;

		10:
			IF TestFBBusy.InitComplete AND NOT TestFBBusy.Busy THEN
				TestFBBusy.Enable();
				State := State + 10;
			END_IF

		20:
			IF TestFBBusy.Enabled THEN
				TestFBBusy.Acceleration := 1000;
				TestFBBusy.Deceleration := 1000;
				TestFBBusy.Velocity		:= 100;
				TestFBBusy.MoveAbsolute(100, TRUE);
				State := State + 10;
			END_IF

		30:
			ActualResult := TestFBBusy.Busy;
			AssertEquals_BOOL(Expected := ExpectedResult, Actual := ActualResult, Message := 'Function Block was not busy when Extending');
			TEST_FINISHED();
			State := State + 10;
	END_CASE

	//Call to FB Cyclic Logic
	TestFBBusy.CyclicLogic();
END_IF
END_METHOD

METHOD CommandInhibited
VAR_INST
	State		   : INT;
	ActualResult   : BOOL;
	ExpectedResult : BOOL := TRUE;
END_VAR
IF TEST_ORDERED('CommandInhibitedAlarm') THEN
	CASE State OF
		0:
			IF TestFBAlarm15.InitComplete THEN
				TestFBAlarm15.Override := 0;
				TestFBAlarm15.MoveAbsolute(100, TRUE);
				State := State + 10;
			END_IF

		10:
			IF TestFBAlarm15.Error OR (TestFBAlarm15.InPosition AND NOT TestFBAlarm15.Busy) THEN
				ActualResult := TestFBAlarm15.BasicAxisAlarms[E_BasicAxis.CommandWhileInhibited].bRaised;
				State		 := State + 10;
			END_IF

		20:
			AssertEquals_BOOL(Expected := ExpectedResult, Actual := ActualResult, Message := 'The alarm was not raised for Command Inhibited Error');
			TEST_FINISHED();
			State := State + 10;
	END_CASE

	TestFBAlarm15.CyclicLogic();
END_IF
END_METHOD

METHOD Init
VAR_INST
	State		   : INT;
	ActualResult   : BOOL;
	ExpectedResult : BOOL := TRUE;
	Timeout		   : TON;
END_VAR
IF TEST_ORDERED('BasicAxisInit') THEN
	CASE State OF
		0:
			Timeout.IN := TRUE;
			State	   := State + 10;

		10:
			IF TestFBInit.InitComplete AND NOT TestFBInit.Busy THEN
				State := State + 10;
			END_IF

			IF Timeout.Q THEN
				State := State + 10;
			END_IF

		20:
			ActualResult := TestFBInit.InitComplete;
			AssertEquals_BOOL(Expected := ExpectedResult, Actual := ActualResult, Message := 'Function Block did not init complete in 2s');
			TEST_FINISHED();
			State := State + 10;
	END_CASE

	//Call to FB Cyclic Logic
	Timeout(PT := T#2S);
	TestFBInit.CyclicLogic();
END_IF
END_METHOD

METHOD MCHaltAlarm
VAR_INST
	State		   : INT;
	ActualResult   : BOOL;
	ExpectedResult : BOOL := TRUE;
	WriteADS	   : FB_WriteAdsSymByName;
END_VAR
IF TEST_ORDERED('MCHaltAlarm') THEN
	CASE State OF
		0:
			WriteADS(bWrite	  := TRUE,
					 sNetId	  := '',
					 nPort	  := 851,
					 sVarName := 'PRG_TEST.ComponentBasicAxisTest.TestFBAlarm4.BasicAxis.MCHalt.Error',
					 nSrcAddr := ADR(ExpectedResult),
					 nLen	  := SIZEOF(ExpectedResult),
					 tTimeout := T#2S,
					 eComMode :=,
					 bBusy	  =>,
					 bError	  =>,
					 nErrorId =>);

			IF NOT WriteADS.bBusy OR WriteADS.bError THEN
				State := State + 10;
			END_IF

			IF TestFBAlarm4.BasicAxisAlarms[E_BasicAxis.HaltError].bRaised THEN
				ActualResult := TestFBAlarm4.BasicAxisAlarms[E_BasicAxis.HaltError].bRaised;
				State		 := State + 10;
			END_IF

		10:
			AssertEquals_BOOL(Expected := ExpectedResult, Actual := ActualResult, Message := 'The alarm was not raised for MC_Halt.Error');
			TEST_FINISHED();
			State := State + 10;
	END_CASE

	TestFBAlarm4.CyclicLogic();
END_IF
END_METHOD

METHOD MCHomeAlarm
VAR_INST
	State		   : INT;
	ActualResult   : BOOL;
	ExpectedResult : BOOL := TRUE;
	WriteADS	   : FB_WriteAdsSymByName;
END_VAR
IF TEST_ORDERED('MCHomeAlarm') THEN
	CASE State OF
		0:
			WriteADS(bWrite	  := TRUE,
					 sNetId	  := '',
					 nPort	  := 851,
					 sVarName := 'PRG_TEST.ComponentBasicAxisTest.TestFBAlarm6.BasicAxis.DefaultHome._Error',
					 nSrcAddr := ADR(ExpectedResult),
					 nLen	  := SIZEOF(ExpectedResult),
					 tTimeout := T#2S,
					 eComMode :=,
					 bBusy	  =>,
					 bError	  =>,
					 nErrorId =>);

			IF NOT WriteADS.bBusy OR WriteADS.bError THEN
				State := State + 10;
			END_IF

			IF TestFBAlarm6.BasicAxisAlarms[E_BasicAxis.HomeError].bRaised THEN
				ActualResult := TestFBAlarm6.BasicAxisAlarms[E_BasicAxis.HomeError].bRaised;
				State		 := State + 10;
			END_IF

		10:
			AssertEquals_BOOL(Expected := ExpectedResult, Actual := ActualResult, Message := 'The alarm was not raised for HomeMethod.Error');
			TEST_FINISHED();
			State := State + 10;
	END_CASE

	TestFBAlarm6.CyclicLogic();
END_IF
END_METHOD

METHOD MCJogAlarm
VAR_INST
	State		   : INT;
	ActualResult   : BOOL;
	ExpectedResult : BOOL := TRUE;
	WriteADS	   : FB_WriteAdsSymByName;
END_VAR
IF TEST_ORDERED('MCJogAlarm') THEN
	CASE State OF
		0:
			WriteADS(bWrite	  := TRUE,
					 sNetId	  := '',
					 nPort	  := 851,
					 sVarName := 'PRG_TEST.ComponentBasicAxisTest.TestFBAlarm7.BasicAxis.MCJog.Error',
					 nSrcAddr := ADR(ExpectedResult),
					 nLen	  := SIZEOF(ExpectedResult),
					 tTimeout := T#2S,
					 eComMode :=,
					 bBusy	  =>,
					 bError	  =>,
					 nErrorId =>);

			IF NOT WriteADS.bBusy OR WriteADS.bError THEN
				State := State + 10;
			END_IF

			IF TestFBAlarm7.BasicAxisAlarms[E_BasicAxis.JogError].bRaised THEN
				ActualResult := TestFBAlarm7.BasicAxisAlarms[E_BasicAxis.JogError].bRaised;
				State		 := State + 10;
			END_IF

		10:
			AssertEquals_BOOL(Expected := ExpectedResult, Actual := ActualResult, Message := 'The alarm was not raised for MCJog.Error');
			TEST_FINISHED();
			State := State + 10;
	END_CASE

	TestFBAlarm7.CyclicLogic();
END_IF
END_METHOD

METHOD MCMoveAbsoluteAlarm
VAR_INST
	State		   : INT;
	ActualResult   : BOOL;
	ExpectedResult : BOOL := TRUE;
END_VAR
IF TEST_ORDERED('MCMoveAbsAlarm') THEN
	CASE State OF
		0:
			IF TestFBAlarm8.InitComplete THEN
				TestFBAlarm8.MoveAbsolute(100, TRUE);
				State := State + 10;
			END_IF

		10:
			IF TestFBAlarm8.Error OR (TestFBAlarm8.InPosition AND NOT TestFBAlarm8.Busy) THEN
				State := State + 10;
			END_IF

		20:
			ActualResult := TestFBAlarm8.BasicAxisAlarms[E_BasicAxis.MoveAbsoluteError].bRaised;
			AssertEquals_BOOL(Expected := ExpectedResult, Actual := ActualResult, Message := 'The alarm was not raised for Move Absolute Error');
			TEST_FINISHED();
			State := State + 10;
	END_CASE

	TestFBAlarm8.CyclicLogic();
END_IF
END_METHOD

METHOD MCMoveModulo
VAR_INST
	State		   : INT;
	ActualResult   : BOOL;
	ExpectedResult : BOOL := TRUE;
END_VAR
IF TEST_ORDERED('MCMoveModuloAlarm') THEN
	CASE State OF
		0:
			IF TestFBAlarm11.InitComplete THEN
				TestFBAlarm11.MoveModulo(100, MC_Direction.MC_Positive_Direction, TRUE);
				State := State + 10;
			END_IF

		10:
			IF TestFBAlarm11.Error OR (TestFBAlarm11.InPosition AND NOT TestFBAlarm11.Busy) THEN
				State := State + 10;
			END_IF

		20:
			ActualResult := TestFBAlarm11.BasicAxisAlarms[E_BasicAxis.MoveModuloError].bRaised;
			AssertEquals_BOOL(Expected := ExpectedResult, Actual := ActualResult, Message := 'The alarm was not raised for Move Modulo Error');
			TEST_FINISHED();
			State := State + 10;
	END_CASE

	TestFBAlarm11.CyclicLogic();
END_IF
END_METHOD

METHOD MCMoveRelativeAlarm
VAR_INST
	State		   : INT;
	ActualResult   : BOOL;
	ExpectedResult : BOOL := TRUE;
END_VAR
IF TEST_ORDERED('MCMoveAbsAlarm') THEN
	CASE State OF
		0:
			IF TestFBAlarm9.InitComplete THEN
				TestFBAlarm9.MoveRelative(100, TRUE);
				State := State + 10;
			END_IF

		10:
			IF TestFBAlarm9.Error OR (TestFBAlarm9.InPosition AND NOT TestFBAlarm9.Busy) THEN
				State := State + 10;
			END_IF

		20:
			ActualResult := TestFBAlarm9.BasicAxisAlarms[E_BasicAxis.MoveRelativeError].bRaised;
			AssertEquals_BOOL(Expected := ExpectedResult, Actual := ActualResult, Message := 'The alarm was not raised for Move Relative Error');
			TEST_FINISHED();
			State := State + 10;
	END_CASE

	TestFBAlarm9.CyclicLogic();
END_IF
END_METHOD

METHOD MCMoveVelocity
VAR_INST
	State		   : INT;
	ActualResult   : BOOL;
	ExpectedResult : BOOL := TRUE;
END_VAR
IF TEST_ORDERED('MCMoveVelAlarm') THEN
	CASE State OF
		0:
			IF TestFBAlarm10.InitComplete THEN
				TestFBAlarm10.MoveVelocity(100, TRUE);
				State := State + 10;
			END_IF

		10:
			IF TestFBAlarm10.Error OR (TestFBAlarm10.InPosition AND NOT TestFBAlarm10.Busy) THEN
				State := State + 10;
			END_IF

		20:
			ActualResult := TestFBAlarm10.BasicAxisAlarms[E_BasicAxis.MoveVelocityError].bRaised;
			AssertEquals_BOOL(Expected := ExpectedResult, Actual := ActualResult, Message := 'The alarm was not raised for Move Relative Error');
			TEST_FINISHED();
			State := State + 10;
	END_CASE

	TestFBAlarm10.CyclicLogic();
END_IF
END_METHOD

METHOD MCPowerAlarm
VAR_INST
	State		   : INT;
	ActualResult   : BOOL;
	ExpectedResult : BOOL := TRUE;
	WriteADS	   : FB_WriteAdsSymByName;
END_VAR
IF TEST_ORDERED('MCPowerAlarm') THEN
	CASE State OF
		0:
			WriteADS(bWrite	  := TRUE,
					 sNetId	  := '',
					 nPort	  := 851,
					 sVarName := 'PRG_TEST.ComponentBasicAxisTest.TestFBAlarm2.BasicAxis.MCPower.Error',
					 nSrcAddr := ADR(ExpectedResult),
					 nLen	  := SIZEOF(ExpectedResult),
					 tTimeout := T#2S,
					 eComMode :=,
					 bBusy	  =>,
					 bError	  =>,
					 nErrorId =>);

			IF NOT WriteADS.bBusy OR WriteADS.bError THEN
				State := State + 10;
			END_IF

			IF TestFBAlarm2.BasicAxisAlarms[E_BasicAxis.PowerError].bRaised THEN
				ActualResult := TestFBAlarm2.BasicAxisAlarms[E_BasicAxis.PowerError].bRaised;
				State		 := State + 10;
			END_IF

		10:
			AssertEquals_BOOL(Expected := ExpectedResult, Actual := ActualResult, Message := 'The alarm was not raised for MC_Power.Error');
			TEST_FINISHED();
			State := State + 10;
	END_CASE

	TestFBAlarm2.CyclicLogic();
END_IF
END_METHOD

METHOD McReadAxisParametersAlarm
VAR_INST
	State		   : INT;
	ActualResult   : BOOL;
	ExpectedResult : BOOL := TRUE;
	WriteADS	   : FB_WriteAdsSymByName;
END_VAR
IF TEST_ORDERED('MCReadAxisAlarm') THEN
	CASE State OF
		0:
			WriteADS(bWrite	  := TRUE,
					 sNetId	  := '',
					 nPort	  := 851,
					 sVarName := 'PRG_TEST.ComponentBasicAxisTest.TestFBAlarm12.BasicAxis.MCReadParameterSet.Error',
					 nSrcAddr := ADR(ExpectedResult),
					 nLen	  := SIZEOF(ExpectedResult),
					 tTimeout := T#2S,
					 eComMode :=,
					 bBusy	  =>,
					 bError	  =>,
					 nErrorId =>);

			IF NOT WriteADS.bBusy OR WriteADS.bError THEN
				State := State + 10;
			END_IF

			IF TestFBAlarm12.BasicAxisAlarms[E_BasicAxis.ReadParameterSetError].bRaised THEN
				ActualResult := TestFBAlarm12.BasicAxisAlarms[E_BasicAxis.ReadParameterSetError].bRaised;
				State		 := State + 10;
			END_IF

		10:
			AssertEquals_BOOL(Expected := ExpectedResult, Actual := ActualResult, Message := 'The alarm was not raised for MC Read Axis Parameter Error');
			TEST_FINISHED();
			State := State + 10;
	END_CASE

	TestFBAlarm12.CyclicLogic();
END_IF
END_METHOD

METHOD MCResetAlarm
VAR_INST
	State		   : INT;
	ActualResult   : BOOL;
	ExpectedResult : BOOL := TRUE;
	WriteADS	   : FB_WriteAdsSymByName;
END_VAR
IF TEST_ORDERED('MCResetAlarm') THEN
	CASE State OF
		0:
			WriteADS(bWrite	  := TRUE,
					 sNetId	  := '',
					 nPort	  := 851,
					 sVarName := 'PRG_TEST.ComponentBasicAxisTest.TestFBAlarm3.BasicAxis.DefaultReset._Error',
					 nSrcAddr := ADR(ExpectedResult),
					 nLen	  := SIZEOF(ExpectedResult),
					 tTimeout := T#2S,
					 eComMode :=,
					 bBusy	  =>,
					 bError	  =>,
					 nErrorId =>);

			IF NOT WriteADS.bBusy OR WriteADS.bError THEN
				State := State + 10;
			END_IF

			IF TestFBAlarm3.BasicAxisAlarms[E_BasicAxis.ResetError].bRaised THEN
				ActualResult := TestFBAlarm3.BasicAxisAlarms[E_BasicAxis.ResetError].bRaised;
				State		 := State + 10;
			END_IF

		10:
			AssertEquals_BOOL(Expected := ExpectedResult, Actual := ActualResult, Message := 'The alarm was not raised for ResetMethod.Error');
			TEST_FINISHED();
			State := State + 10;
	END_CASE

	TestFBAlarm3.CyclicLogic();
END_IF
END_METHOD

METHOD McWriteAxisBoolParameterAlarm
VAR_INST
	State		   : INT;
	ActualResult   : BOOL;
	ExpectedResult : BOOL := TRUE;
	WriteADS	   : FB_WriteAdsSymByName;
END_VAR
IF TEST_ORDERED('MCWriteAxisBoolAlarm') THEN
	CASE State OF
		0:
			WriteADS(bWrite	  := TRUE,
					 sNetId	  := '',
					 nPort	  := 851,
					 sVarName := 'PRG_TEST.ComponentBasicAxisTest.TestFBAlarm14.BasicAxis.MCWriteBoolParameter.Error',
					 nSrcAddr := ADR(ExpectedResult),
					 nLen	  := SIZEOF(ExpectedResult),
					 tTimeout := T#2S,
					 eComMode :=,
					 bBusy	  =>,
					 bError	  =>,
					 nErrorId =>);

			IF NOT WriteADS.bBusy OR WriteADS.bError THEN
				State := State + 10;
			END_IF

			IF TestFBAlarm14.BasicAxisAlarms[E_BasicAxis.WriteBoolParameterError].bRaised THEN
				ActualResult := TestFBAlarm14.BasicAxisAlarms[E_BasicAxis.WriteBoolParameterError].bRaised;
				State		 := State + 10;
			END_IF

		10:
			AssertEquals_BOOL(Expected := ExpectedResult, Actual := ActualResult, Message := 'The alarm was not raised for MC Write Axis Bool Parameter Error');
			TEST_FINISHED();
			State := State + 10;
	END_CASE

	TestFBAlarm14.CyclicLogic();
END_IF
END_METHOD

METHOD McWriteAxisParameterAlarm
VAR_INST
	State		   : INT;
	ActualResult   : BOOL;
	ExpectedResult : BOOL := TRUE;
	WriteADS	   : FB_WriteAdsSymByName;
END_VAR
IF TEST_ORDERED('MCWriteAxisAlarm') THEN
	CASE State OF
		0:
			WriteADS(bWrite	  := TRUE,
					 sNetId	  := '',
					 nPort	  := 851,
					 sVarName := 'PRG_TEST.ComponentBasicAxisTest.TestFBAlarm13.BasicAxis.MCWriteParameter.Error',
					 nSrcAddr := ADR(ExpectedResult),
					 nLen	  := SIZEOF(ExpectedResult),
					 tTimeout := T#2S,
					 eComMode :=,
					 bBusy	  =>,
					 bError	  =>,
					 nErrorId =>);

			IF NOT WriteADS.bBusy OR WriteADS.bError THEN
				State := State + 10;
			END_IF

			IF TestFBAlarm13.BasicAxisAlarms[E_BasicAxis.WriteParameterError].bRaised THEN
				ActualResult := TestFBAlarm13.BasicAxisAlarms[E_BasicAxis.WriteParameterError].bRaised;
				State		 := State + 10;
			END_IF

		10:
			AssertEquals_BOOL(Expected := ExpectedResult, Actual := ActualResult, Message := 'The alarm was not raised for MC Write Axis Parameter Error');
			TEST_FINISHED();
			State := State + 10;
	END_CASE

	TestFBAlarm13.CyclicLogic();
END_IF
END_METHOD

METHOD NameSetProperty
VAR_INST
	State			: INT;
	ActualResult	: STRING;
	ActualResultHMI : STRING;
	ExpectedResult	: STRING := 'TEST_NAME';
END_VAR
IF TEST_ORDERED('BasicAxisNameSetProperty') THEN
	CASE State OF
		0:
			State := State + 10;

		10:
			IF TestFBNameSetProperty.InitComplete AND NOT TestFBNameSetProperty.Busy THEN
				State := State + 10;
			END_IF

		20:
			TestFBNameSetProperty.Name := ExpectedResult;
			State					   := State + 10;

		30:
			ActualResultHMI := TestFBNameSetProperty.ComponentBase_HMI.Config.Name;
			ActualResult	:= TestFBNameSetProperty.Name;
			AssertEquals(Expected := ExpectedResult, Actual := ActualResult, Message := 'Name was not read by Property correctly');
			AssertEquals(Expected := ExpectedResult, Actual := ActualResultHMI, Message := 'Name was not read by HMI correctly');
			TEST_FINISHED();
			State := State + 10;
	END_CASE

	//Call to FB Cyclic Logic
	TestFBNameSetProperty.CyclicLogic();
END_IF
END_METHOD

METHOD SimulationCheckAlarm
VAR_INST
	State		   : INT;
	ActualResult   : BOOL;
	ExpectedResult : BOOL := TRUE;
END_VAR
IF TEST_ORDERED('BasicAxisSimulationCheckAlarm') THEN
	CASE State OF
		0:
			State := State + 10;

		10:
			IF TestFBSimulationCheckAlarm.InitComplete AND NOT TestFBSimulationCheckAlarm.Busy THEN
				State := State + 10;
			END_IF

		20:
			TestFBSimulationCheckAlarm.InSimulation := TRUE; //Set simulation to true;
			State									:= State + 10;

		30:
			ActualResult := TestFBSimulationCheckAlarm.ComponentBaseAlarms[E_ComponentBase.SimulationWarning].bRaised;
			AssertEquals_BOOL(Expected := ExpectedResult, Actual := ActualResult, Message := 'Function Block did Raise alarm when in simulation');
			TEST_FINISHED();
			State := State + 10;
	END_CASE

	//Call to FB Cyclic Logic
	TestFBSimulationCheckAlarm.CyclicLogic();
END_IF
END_METHOD

METHOD SimulationSetHMI
VAR_INST
	State			: INT;
	ActualResult	: BOOL;
	ActualResultHMI : BOOL;
	ExpectedResult	: BOOL := TRUE;
	WriteADS		: FB_WriteAdsSymByName;
END_VAR
IF TEST_ORDERED('BasicAxisSetSimulationHMI') THEN
	CASE State OF
		0:
			State := State + 10;

		10:
			IF TestFBSimulationSetHMI.InitComplete AND NOT TestFBSimulationSetHMI.Busy THEN
				TestFBSimulationSetHMI.AllowHMIControl(); // Must turn on Allow control for code to function
				State := State + 10;
			END_IF

		20:
			WriteADS(bWrite	  := TRUE,
					 sNetId	  := '',
					 nPort	  := 851,
					 sVarName := 'PRG_TEST.ComponentBasicAxisTest.TestFBSimulationSetHMI.ComponentBase_HMI.Command.SimulatedOperation',
					 nSrcAddr := ADR(ExpectedResult),
					 nLen	  := SIZEOF(ExpectedResult),
					 tTimeout := T#2S,
					 eComMode :=,
					 bBusy	  =>,
					 bError	  =>,
					 nErrorId =>);

			IF NOT WriteADS.bBusy OR WriteADS.bError THEN
				State := State + 10;
			END_IF

		30:
			ActualResult	:= TestFBSimulationSetHMI.InSimulation;
			ActualResultHMI := TestFBSimulationSetHMI.ComponentBase_HMI.Status.InSimulation;
			AssertEquals_BOOL(Expected := ExpectedResult, Actual := ActualResult, Message := 'Function Block did not set simulation by HMI when read by Property');
			AssertEquals_BOOL(Expected := ExpectedResult, Actual := ActualResultHMI, Message := 'Function Block did not set simulation by HMI when read by HMI');
			TEST_FINISHED();
			State := State + 10;
	END_CASE

	//Call to FB Cyclic Logic
	TestFBSimulationSetHMI.CyclicLogic();
END_IF
END_METHOD

METHOD SimulationSetProperty
VAR_INST
	State			: INT;
	ActualResult	: BOOL;
	ActualResultHMI : BOOL;
	ExpectedResult	: BOOL := TRUE;
END_VAR
IF TEST_ORDERED('BasicAxisSetSimulationProperty') THEN
	CASE State OF
		0:
			State := State + 10;

		10:
			IF TestFBSimulationSetProperty.InitComplete AND NOT TestFBSimulationSetProperty.Busy THEN
				State := State + 10;
			END_IF

		20:
			TestFBSimulationSetProperty.InSimulation := TRUE;
			State									 := State + 10;

		30:
			ActualResult	:= TestFBSimulationSetProperty.InSimulation;
			ActualResultHMI := TestFBSimulationSetProperty.ComponentBase_HMI.Status.InSimulation;
			AssertEquals_BOOL(Expected := ExpectedResult, Actual := ActualResult, Message := 'Function Block did not set simulation by property when read by Property');
			AssertEquals_BOOL(Expected := ExpectedResult, Actual := ActualResultHMI, Message := 'Function Block did not set simulation by property when read by HMI');
			TEST_FINISHED();
			State := State + 10;
	END_CASE

	//Call to FB Cyclic Logic
	TestFBSimulationSetProperty.CyclicLogic();
END_IF
END_METHOD

END_FUNCTION_BLOCK

// Testing/PRG_TEST
PROGRAM PRG_TEST
VAR
	SingleSolenoidTest		   : FB_SingleSolenoid_Test;
	DoubleSolenoidTest		   : FB_DoubleSolenoid_Test;
	SingleSolenoidFeedbackTest : FB_SingleSolenoidFeedback_Test;
	ComponentBasicAxisTest	   : FB_ComponentBasicAxis_Test;
	PlcTaskComponent		   : FB_PlcCameraBase;
	visionTaskComponent		   : FB_VisionCameraDetection;
END_VAR

TcUnit.RUN();



PlcTaskComponent.RunVision := TRUE;

END_PROGRAM

// Testing/Solenoids/FB_SingleSolenoid_Test
FUNCTION_BLOCK FB_SingleSolenoid_Test EXTENDS TcUnit.FB_TestSuite
VAR
	// FBs for ComponentBase
	TestFBInit					: FB_SingleSolenoid;
	TestFBNameSetProperty		: FB_SingleSolenoid;
	TestFBNameSetHMI			: FB_SingleSolenoid;
	TestFBSimulationSetProperty : FB_SingleSolenoid;
	TestFBSimulationSetHMI		: FB_SingleSolenoid;
	TestFBSimulationCheckAlarm	: FB_SingleSolenoid;
	TestFBBusy					: FB_SingleSolenoid;
	TestFBAllowHMI				: FB_SingleSolenoid;
	TestFBBlockHMI				: FB_SingleSolenoid;

	// Solenoid FB	
	TestSingleSolenoidExtend  : FB_SingleSolenoid;
	TestSingleSolenoidRetract : FB_SingleSolenoid;
END_VAR

Init();
NameSetProperty();
SimulationSetProperty();
SimulationSetHMI();
SimulationCheckAlarm();
Busy();
AllowHMI();
BlockHMI();
ExtendEqualsExtendedOutputOn();
RetractEqualsExtendOutputOff();

METHOD AllowHMI
VAR_INST
	State		   : INT;
	ActualResult   : BOOL;
	ExpectedResult : BOOL := TRUE;
END_VAR
IF TEST_ORDERED('AllowHMI') THEN
	CASE State OF
		0:
			State := State + 10;

		10:
			IF TestFBAllowHMI.InitComplete AND NOT TestFBAllowHMI.Busy THEN
				TestFBAllowHMI.AllowHMIControl();
				State := State + 10;
			END_IF

		20:
			ActualResult := TestFBAllowHMI.ComponentBase_HMI.Status.HMIControlAvailable;
			AssertEquals_BOOL(Expected := ExpectedResult, Actual := ActualResult, Message := 'Function Block read allow HMI Control in HMI Tag not true');
			TEST_FINISHED();
			State := State + 10;
	END_CASE

	//Call to FB Cyclic Logic
	TestFBAllowHMI.CyclicLogic();
END_IF
END_METHOD

METHOD BlockHMI
VAR_INST
	State		   : INT;
	ActualResult   : BOOL;
	ExpectedResult : BOOL := FALSE;
END_VAR
IF TEST_ORDERED('BlockHMI') THEN
	CASE State OF
		0:
			State := State + 10;

		10:
			IF TestFBBlockHMI.InitComplete AND NOT TestFBBlockHMI.Busy THEN
				TestFBBlockHMI.AllowHMIControl();
				State := State + 10;
			END_IF

		20:
			IF TestFBBlockHMI.ComponentBase_HMI.Status.HMIControlAvailable THEN
				TestFBBlockHMI.BlockHMIControl();
				State := State + 10;
			END_IF

		30:
			ActualResult := TestFBBlockHMI.ComponentBase_HMI.Status.HMIControlAvailable;
			AssertEquals_BOOL(Expected := ExpectedResult, Actual := ActualResult, Message := 'Function Block read Block HMI Control in HMI Tag not false');
			TEST_FINISHED();
			State := State + 10;
	END_CASE

	//Call to FB Cyclic Logic
	TestFBBlockHMI.CyclicLogic();
END_IF
END_METHOD

METHOD Busy
VAR_INST
	State		   : INT;
	ActualResult   : BOOL;
	ExpectedResult : BOOL := TRUE;
	Timeout		   : TON;
END_VAR
IF TEST_ORDERED('Busy') THEN
	CASE State OF
		0:
			State := State + 10;

		10:
			IF TestFBBusy.InitComplete AND NOT TestFBBusy.Busy THEN
				State := State + 10;
			END_IF

		20:
			TestFBBusy.Extend();
			State := State + 10;

		30:
			ActualResult := TestFBBusy.Busy;
			AssertEquals_BOOL(Expected := ExpectedResult, Actual := ActualResult, Message := 'Function Block was not busy when Extending');
			TEST_FINISHED();
			State := State + 10;
	END_CASE

	//Call to FB Cyclic Logic
	TestFBBusy.CyclicLogic();
END_IF
END_METHOD

METHOD ExtendEqualsExtendedOutputOn
VAR_INST
	State		   : INT;
	ActualResult   : BOOL;
	ExpectedResult : BOOL := TRUE;
END_VAR
IF TEST_ORDERED('ExtendEqualsExtendedOutputOn') THEN
	CASE State OF
		0:
			State := State + 10;

		10:
			TestSingleSolenoidExtend.Extend();
			State := State + 10;

		20:
			ActualResult := TestSingleSolenoidExtend.ExtendOutput;
			AssertEquals_BOOL(Expected := ExpectedResult, Actual := ActualResult, Message := 'Solenoid did not set output on');
			TEST_FINISHED();
			State := State + 10;
	END_CASE

	TestSingleSolenoidExtend.CyclicLogic();
END_IF
END_METHOD

METHOD Init
VAR_INST
	State		   : INT;
	ActualResult   : BOOL;
	ExpectedResult : BOOL := TRUE;
	Timeout		   : TON;
END_VAR
IF TEST_ORDERED('Init') THEN
	CASE State OF
		0:
			Timeout.IN := TRUE;
			State	   := State + 10;

		10:
			IF TestFBInit.InitComplete AND NOT TestFBInit.Busy THEN
				State := State + 10;
			END_IF

			IF Timeout.Q THEN
				State := State + 10;
			END_IF

		20:
			ActualResult := TestFBInit.InitComplete;
			AssertEquals_BOOL(Expected := ExpectedResult, Actual := ActualResult, Message := 'Function Block did not init complete in 2s');
			TEST_FINISHED();
			State := State + 10;
	END_CASE

	//Call to FB Cyclic Logic
	Timeout(PT := T#2S);
	TestFBInit.CyclicLogic();
END_IF
END_METHOD

METHOD NameSetProperty
VAR_INST
	State			: INT;
	ActualResult	: STRING;
	ActualResultHMI : STRING;
	ExpectedResult	: STRING := 'TEST_NAME';
END_VAR
IF TEST_ORDERED('NameSetProperty') THEN
	CASE State OF
		0:
			State := State + 10;

		10:
			IF TestFBNameSetProperty.InitComplete AND NOT TestFBNameSetProperty.Busy THEN
				State := State + 10;
			END_IF

		20:
			TestFBNameSetProperty.Name := ExpectedResult;
			State					   := State + 10;

		30:
			ActualResultHMI := TestFBNameSetProperty.ComponentBase_HMI.Config.Name;
			ActualResult	:= TestFBNameSetProperty.Name;
			AssertEquals(Expected := ExpectedResult, Actual := ActualResult, Message := 'Name was not read by Property correctly');
			AssertEquals(Expected := ExpectedResult, Actual := ActualResultHMI, Message := 'Name was not read by HMI correctly');
			TEST_FINISHED();
			State := State + 10;
	END_CASE

	//Call to FB Cyclic Logic
	TestFBNameSetProperty.CyclicLogic();
END_IF
END_METHOD

METHOD RetractEqualsExtendOutputOff
VAR_INST
	State		   : INT;
	ActualResult   : BOOL;
	ExpectedResult : BOOL := FALSE;
END_VAR
IF TEST_ORDERED('RetractEqualsExtendOutputOff') THEN
	CASE State OF
		0:
			State := State + 10;

		10:
			TestSingleSolenoidRetract.Retract();
			State := State + 10;

		20:
			ActualResult := TestSingleSolenoidRetract.ExtendOutput;
			AssertEquals_BOOL(Expected := ExpectedResult, Actual := ActualResult, Message := 'Solenoid did not set output on');
			TEST_FINISHED();
			State := State + 10;
	END_CASE

	TestSingleSolenoidRetract.CyclicLogic();
END_IF
END_METHOD

METHOD SimulationCheckAlarm
VAR_INST
	State		   : INT;
	ActualResult   : BOOL;
	ExpectedResult : BOOL := TRUE;
END_VAR
IF TEST_ORDERED('SimulationCheckAlarm') THEN
	CASE State OF
		0:
			State := State + 10;

		10:
			IF TestFBSimulationCheckAlarm.InitComplete AND NOT TestFBSimulationCheckAlarm.Busy THEN
				State := State + 10;
			END_IF

		20:
			TestFBSimulationCheckAlarm.InSimulation := TRUE; //Set simulation to true;
			State									:= State + 10;

		30:
			ActualResult := TestFBSimulationCheckAlarm.ComponentBaseAlarms[E_ComponentBase.SimulationWarning].bRaised;
			AssertEquals_BOOL(Expected := ExpectedResult, Actual := ActualResult, Message := 'Function Block did Raise alarm when in simulation');
			TEST_FINISHED();
			State := State + 10;
	END_CASE

	//Call to FB Cyclic Logic
	TestFBSimulationCheckAlarm.CyclicLogic();
END_IF
END_METHOD

METHOD SimulationSetHMI
VAR_INST
	State			: INT;
	ActualResult	: BOOL;
	ActualResultHMI : BOOL;
	ExpectedResult	: BOOL := TRUE;
	WriteADS		: FB_WriteAdsSymByName;
END_VAR
IF TEST_ORDERED('SimulationSetHMI') THEN
	CASE State OF
		0:
			State := State + 10;

		10:
			IF TestFBSimulationSetHMI.InitComplete AND NOT TestFBSimulationSetHMI.Busy THEN
				TestFBSimulationSetHMI.AllowHMIControl(); // Must turn on Allow control for code to function
				State := State + 10;
			END_IF

		20:
			WriteADS(bWrite	  := TRUE,
					 sNetId	  := '',
					 nPort	  := 851,
					 sVarName := 'PRG_TEST.SingleSolenoidTest.TestFBSimulationSetHMI.ComponentBase_HMI.Command.SimulatedOperation',
					 nSrcAddr := ADR(ExpectedResult),
					 nLen	  := SIZEOF(ExpectedResult),
					 tTimeout := T#2S,
					 eComMode :=,
					 bBusy	  =>,
					 bError	  =>,
					 nErrorId =>);

			IF NOT WriteADS.bBusy OR WriteADS.bError THEN
				State := State + 10;
			END_IF

		30:
			ActualResult	:= TestFBSimulationSetHMI.InSimulation;
			ActualResultHMI := TestFBSimulationSetHMI.ComponentBase_HMI.Status.InSimulation;
			AssertEquals_BOOL(Expected := ExpectedResult, Actual := ActualResult, Message := 'Function Block did not set simulation by HMI when read by Property');
			AssertEquals_BOOL(Expected := ExpectedResult, Actual := ActualResultHMI, Message := 'Function Block did not set simulation by HMI when read by HMI');
			TEST_FINISHED();
			State := State + 10;
	END_CASE

	//Call to FB Cyclic Logic
	TestFBSimulationSetHMI.CyclicLogic();
END_IF
END_METHOD

METHOD SimulationSetProperty
VAR_INST
	State			: INT;
	ActualResult	: BOOL;
	ActualResultHMI : BOOL;
	ExpectedResult	: BOOL := TRUE;
END_VAR
IF TEST_ORDERED('SimulationSetProperty') THEN
	CASE State OF
		0:
			State := State + 10;

		10:
			IF TestFBSimulationSetProperty.InitComplete AND NOT TestFBSimulationSetProperty.Busy THEN
				State := State + 10;
			END_IF

		20:
			TestFBSimulationSetProperty.InSimulation := TRUE;
			State									 := State + 10;

		30:
			ActualResult	:= TestFBSimulationSetProperty.InSimulation;
			ActualResultHMI := TestFBSimulationSetProperty.ComponentBase_HMI.Status.InSimulation;
			AssertEquals_BOOL(Expected := ExpectedResult, Actual := ActualResult, Message := 'Function Block did not set simulation by property when read by Property');
			AssertEquals_BOOL(Expected := ExpectedResult, Actual := ActualResultHMI, Message := 'Function Block did not set simulation by property when read by HMI');
			TEST_FINISHED();
			State := State + 10;
	END_CASE

	//Call to FB Cyclic Logic
	TestFBSimulationSetProperty.CyclicLogic();
END_IF
END_METHOD

END_FUNCTION_BLOCK

// Testing/Solenoids/FB_DoubleSolenoid_Test
FUNCTION_BLOCK FB_DoubleSolenoid_Test EXTENDS TcUnit.FB_TestSuite
VAR
	TestFBExtend  : FB_DoubleSolenoid;
	TestFBRetract : FB_DoubleSolenoid;
END_VAR

ExtendEqualsExtendOutputOnRetractOff();
RetractEqualsExtendOutputOffRetractOutputOn();

METHOD ExtendEqualsExtendOutputOnRetractOff
VAR_INST
	State						: INT;
	ActualExtendOutputResult	: BOOL;
	ActualRetractOutputResult	: BOOL;
	ExpectedExtendOutputResult	: BOOL := TRUE;
	ExpectedRetractOutputResult : BOOL := FALSE;
END_VAR
IF TEST_ORDERED('ExtendEqualsExtendOutputOnRetractOff') THEN
	CASE State OF
		0:
			State := State + 10;

		10:
			IF TestFBExtend.InitComplete AND NOT TestFBExtend.Busy THEN
				TestFBExtend.Extend();
				State := State + 10;
			END_IF

		20:
			ActualExtendOutputResult := TestFBExtend.ExtendOutput;
			AssertEquals_BOOL(Expected := ExpectedExtendOutputResult, Actual := ActualExtendOutputResult, Message := 'Solenoid did not set extend output on');
			ActualRetractOutputResult := TestFBExtend.RetractOutput;
			AssertEquals_BOOL(Expected := ExpectedRetractOutputResult, Actual := ActualRetractOutputResult, Message := 'Solenoid did not set retract output off');
			TEST_FINISHED();
			State := State + 10;
	END_CASE

	TestFBExtend.CyclicLogic();
END_IF
END_METHOD

METHOD RetractEqualsExtendOutputOffRetractOutputOn
VAR_INST
	State						: INT;
	ActualExtendOutputResult	: BOOL;
	ActualRetractOutputResult	: BOOL;
	ExpectedExtendOutputResult	: BOOL := FALSE;
	ExpectedRetractOutputResult : BOOL := TRUE;
END_VAR
IF TEST_ORDERED('ExtendEqualsExtendOutputOffRetractOn') THEN
	CASE State OF
		0:
			State := State + 10;

		10:
			IF TestFBRetract.InitComplete AND NOT TestFBRetract.Busy THEN
				TestFBRetract.Extend();
				State := State + 10;
			END_IF

		20:
			IF TestFBRetract.Extended THEN
				TestFBRetract.Retract();
				State := State + 10;
			END_IF

		30:
			ActualExtendOutputResult := TestFBRetract.ExtendOutput;
			AssertEquals_BOOL(Expected := ExpectedExtendOutputResult, Actual := ActualExtendOutputResult, Message := 'Solenoid did not set extend output off');
			ActualRetractOutputResult := TestFBRetract.RetractOutput;
			AssertEquals_BOOL(Expected := ExpectedRetractOutputResult, Actual := ActualRetractOutputResult, Message := 'Solenoid did not set retract output on');
			TEST_FINISHED();
			State := State + 10;
	END_CASE

	TestFBRetract.CyclicLogic();
END_IF
END_METHOD

END_FUNCTION_BLOCK

// Testing/Solenoids/FB_SingleSolenoidFeedback_Test
FUNCTION_BLOCK FB_SingleSolenoidFeedback_Test EXTENDS FB_TestSuite
VAR
	// Solenoid FB	
	TestSingleSolenoidFeedbackExtend	   : FB_SingleSolenoidFeedback;
	TestSingleSolenoidFeedbackExtendError  : FB_SingleSolenoidFeedback;
	TestSingleSolenoidFeedbackRetract	   : FB_SingleSolenoidFeedback;
	TestSingleSolenoidFeedbackRetractError : FB_SingleSolenoidFeedback;
END_VAR

Extend();
ExtendError();

METHOD Extend
VAR_INST
	State		   : INT;
	ActualResult   : BOOL;
	ExpectedResult : BOOL := TRUE;
END_VAR
IF TEST_ORDERED('SingleSolenoidFeedbackTestExtend') THEN
	CASE State OF
		0:
			IF TestSingleSolenoidFeedbackExtend.InitComplete AND NOT TestSingleSolenoidFeedbackExtend.Busy THEN
				TestSingleSolenoidFeedbackExtend.Extend();
				TestSingleSolenoidFeedbackExtend.ExtendedInput	:= TRUE;  //Set the feedback
				TestSingleSolenoidFeedbackExtend.RetractedInput := FALSE; //Set the feedback
				State											:= State + 10;
			END_IF

		10:
			ActualResult := TestSingleSolenoidFeedbackExtend.Extended;
			AssertEquals_BOOL(Expected := ExpectedResult, Actual := ActualResult, Message := 'Solenoid feedback did not turn on');
			State := State + 10;
			TEST_FINISHED();
	END_CASE

	TestSingleSolenoidFeedbackExtend.CyclicLogic();
END_IF
END_METHOD

METHOD ExtendError
VAR_INST
	State				: INT;
	ActualResult		: BOOL;
	ExpectedResult		: BOOL := FALSE;
	ActualErrorResult	: BOOL;
	ExpectedErrorResult : BOOL := TRUE;
END_VAR
IF TEST_ORDERED('SingleSolenoidFeedbackTestExtendError') THEN
	CASE State OF
		0:
			IF TestSingleSolenoidFeedbackExtendError.InitComplete AND NOT TestSingleSolenoidFeedbackExtendError.Busy THEN
				TestSingleSolenoidFeedbackExtendError.Extend();
				State := State + 10;
			END_IF

		10:
			IF TestSingleSolenoidFeedbackExtendError.Extended OR TestSingleSolenoidFeedbackExtendError.Error THEN
				ActualResult := TestSingleSolenoidFeedbackExtendError.Extended;
				AssertEquals_BOOL(Expected := ExpectedResult, Actual := ActualResult, Message := 'Solenoid feedback did not turn on');
				ActualErrorResult := TestSingleSolenoidFeedbackExtendError.Error;
				AssertEquals_BOOL(Expected := ExpectedErrorResult, Actual := ActualErrorResult, Message := 'Solenoid Feedback extend no error');
				State := State + 10;
				TEST_FINISHED();
			END_IF
	END_CASE

	TestSingleSolenoidFeedbackExtendError.CyclicLogic();
END_IF
END_METHOD

END_FUNCTION_BLOCK

// Vision/PLC Task/FB_PlcCameraBase
FUNCTION_BLOCK FB_PlcCameraBase EXTENDS FB_ComponentBase
VAR
	//Outputs
	SoftwareTrigger	   AT %Q* : BOOL;
	_RunVision		   AT %Q* : BOOL;
	_Reset			   AT %Q* : BOOL;

	//Inputs
	CameraState			 AT %I* : ETcVnCameraState;
	ResultsAvailable	 AT %I* : BOOL;
	NumberOfResults		 AT %I* : UDINT;
	Results				 AT %I* : ARRAY[1..Parameters_Vision.MAX_RESULTS_BUFFER_BYTES] OF BYTE;
	VisionError			 AT %I* : BOOL;
	VisionErrorID		 AT %I* : UDINT;

	
	VisionAlarms : ARRAY[1..5] OF FB_TcAlarm;
END_VAR

//! @summary Initializes event function blocks using this components's name
METHOD PROTECTED CreateEvents

//! @description This method is called by <c>Initialize()</c> as required
SUPER^.CreateEvents();

F_CreateAllEventsInClass(Alarms		:= VisionAlarms,
						 ClassSize	:= SIZEOF(TC_EVENTS.VisionBaseAlarms),
						 pInitEvent := ADR(TC_EVENTS.VisionBaseAlarms.InitReferenceEvent),
						 Prefix		:= Name);
END_METHOD

//! @summary This method serves as the entry point for all underlying FB logic
METHOD PUBLIC CyclicLogic

//! @description This method should be called cyclically by descendant function blocks by invoking <c>SUPER^.CyclicLogic()</c>.  Alternatively, the contents of this method could be reimplemented entirely in which case a call to this method would not be necessary.
SUPER^.CyclicLogic();

// Monitor camera error here
IF VisionError AND NOT VisionAlarms[E_VisionBaseAlarms.CameraFault].bRaised THEN
	VisionAlarms[E_VisionBaseAlarms.CameraFault].Raise(0);
ELSIF NOT VisionError AND VisionAlarms[E_VisionBaseAlarms.CameraFault].bRaised THEN
	VisionAlarms[E_VisionBaseAlarms.CameraFault].Clear(0, 0);
END_IF

_Error := VisionAlarms[E_VisionBaseAlarms.CameraFault].bRaised;
IF _Error THEN
	_ErrorID := VisionErrorID;
//ELSE
//	_ErrorID := 0;
END_IF

_Busy := _RunVision;
END_METHOD

METHOD GetResults : BOOL
VAR_IN_OUT
	ResultArray : ARRAY[1..Parameters_Vision.MAX_RESULTS_BUFFER_BYTES] OF BYTE;
	Number		: UDINT;
END_VAR

VAR_INST
	ResultsAvailable_RTRIG : R_TRIG;
END_VAR
GetResults := FALSE;
ResultsAvailable_RTRIG(CLK := ResultsAvailable);
IF ResultsAvailable_RTRIG.Q THEN
	IF SIZEOF(ResultArray) < SIZEOF(Results) THEN
		MEMCPY(ADR(ResultArray), ADR(Results), SIZEOF(ResultArray));
	ELSE
		MEMCPY(ADR(ResultArray), ADR(Results), SIZEOF(Results));
	END_IF

	IF NumberOfResults * SIZEOF(Results) > SIZEOF(ResultArray) THEN
		; ///Handle alarm
	END_IF

	Number	   := NumberOfResults;
	GetResults := TRUE;
END_IF
END_METHOD

//! @summary Clears error flags and error IDs for this component
METHOD PUBLIC Reset : BOOL
//Return the value from the base FB Reset()
Reset := SUPER^.Reset();

// Clear the Vision Alarms
F_ClearAllEventsInClass(Alarms:=VisionAlarms);

// Set the Error ID to 0
_ErrorID := 0;
END_METHOD

PROPERTY RunVision : BOOL
SET
_RunVision := RunVision;
SoftwareTrigger := false;
END_SET
END_PROPERTY

PROPERTY TriggerImage : BOOL
SET
SoftwareTrigger := TriggerImage;
END_SET
END_PROPERTY

END_FUNCTION_BLOCK

// Vision/VisionTask/FB_VisionCameraDetection
FUNCTION_BLOCK FB_VisionCameraDetection EXTENDS FB_VisionCameraBase
VAR

	// Iterator for Vision
	ipIterator : ITcVnForwardIterator;

	ipContourResultList : ITcVnContainer;
	ipContour			: ITcVnContainer;
	ipResultContainer	: ITcVnContainer;

	// Blob Detection
	///_BlobParams		 : TcVnParamsBlobDetection;
	Offset			 : TcVnPoint;


	//Configuration
	VisionTool : E_VisionTools;


	// Color
	nNewImageCounter : UINT;
	bTrigger		 : BOOL := TRUE;

	// Output
	Text		  : STRING(255);
	NumberOfBlobs : ULINT;
	BlobResults	  : ARRAY[1..100] OF ST_BlobResults;
	
	
END_VAR

METHOD ProcessImage
VAR
	ulint_ref		 : REFERENCE TO ULINT;
	i				 : ULINT;
	Rect			 : TcVnRectangle_UDINT;
	Text			 : STRING;
	Image_ID_NumText : STRING;
	nX				 : UDINT := 20;
	nY				 : UDINT := 50;
END_VAR
SUPER^.ProcessImage();

//Clear Results and set new results-Number of Blobs
MEMSET(ADR(BlobResults), 0, SIZEOF(BlobResults));
MEMSET(ADR(FeedbackResults), 0, SIZEOF(FeedbackResults));
ulint_ref REF= (NumberOfBlobs);
hr		  := F_VN_GetNumberOfElements(ipContainer := ipContourList, nNumberOfElements := ulint_ref, hrPrev := hr);
IF NumberOfBlobs > 0 THEN
	FOR i := 0 TO (NumberOfBlobs - 1) BY 1 DO
		hr := F_VN_GetAt_ITcVnContainer(ipSrcContainer	:= ipContourList,
										ipDestContainer := ipResultContainer,
										nIndex			:= i,
										hrPrev			:= hr);

		hr := F_VN_ContourArea(ipContour := ipResultContainer, fArea := BlobResults[i + 1].Area, hrPrev := hr);
		hr := F_VN_ContourCenterOfMass(ipContour := ipResultContainer, aCenterOfMass := BlobResults[i + 1].CenterOfMass, hrPrev := hr);

		//More items
		hr := F_VN_ContourCircularity(ipContour := ipResultContainer, fCircularity := BlobResults[i + 1].Circularity, hrPrev := hr);
		hr := F_VN_ContourConvexity(ipContour := ipResultContainer, fConvexity := BlobResults[i + 1].Convexity, hrPrev := hr);
		hr := F_VN_ContourEccentricity(ipContour := ipResultContainer, fEccentricity := BlobResults[i + 1].Eccentricity, hrPrev := hr);
		hr := F_VN_ContourInertiaRatio(ipContour := ipResultContainer, fInertiaRatio := BlobResults[i + 1].InertiaRatio, hrPrev := hr);
		hr := F_VN_ContourOrientation(ipContour := ipResultContainer, stOrientation := BlobResults[i + 1].Orientation, hrPrev := hr);
		hr := F_VN_ContourPerimeter(ipContour  := ipResultContainer,
									fPerimeter := BlobResults[i + 1].Perimeter,
									bClosed	   := TRUE,
									hrPrev	   := hr);

		hr := F_VN_ContourRoundness(ipContour := ipResultContainer, fRoundness := BlobResults[i + 1].Roundness, hrPrev := hr);

		//Copy the needed results into the return results
		FeedbackResults[i + 1].x		:= BlobResults[i + 1].CenterOfMass[0];
		FeedbackResults[i + 1].y		:= BlobResults[i + 1].CenterOfMass[1];
		FeedbackResults[i + 1].c		:= BlobResults[i + 1].Orientation.fAngle;
		FeedbackResults[i + 1].Distance := 0;
		FeedbackResults[i + 1].Pass		:= TRUE;
	END_FOR

	//Check the size of the buffer and the size to be copied
	IF SIZEOF(FeedbackResults) < SIZEOF(Results) THEN
		MEMCPY(ADR(Results), ADR(FeedbackResults), SIZEOF(FeedbackResults));
	ELSE
		MEMCPY(ADR(Results), ADR(FeedbackResults), SIZEOF(Results));
	END_IF
END_IF

//Return result number even if none found
NumberOfResults	 := TO_UDINT(NumberOfBlobs);
ResultsAvailable := TRUE;

(* Draw Result Image
// --------------------------------------------------------------*)
hr := F_VN_DrawContours(ipContourList,
						-1,
						ipImageRes,
						GVL_VisionColor.ColorGreen,
						3,
						hr);

IF NumberOfBlobs > 0 THEN
	FOR i := 0 TO (NumberOfBlobs - 1) DO
		hr := F_VN_GetAt_ITcVnContainer(ipSrcContainer	:= ipContourList,
										ipDestContainer := ipResultContainer,
										nIndex			:= i,
										hrPrev			:= hr);

		//hr	 := F_VN_UprightBoundingRectangle(ipResultContainer, Rect, hr);
		Text := TO_STRING(i + 1);
		hr	 := F_VN_PutText(Text,
							 ipImageRes,
							 TO_UDINT(BlobResults[i + 1].CenterOfMass[0]) - 20,
							 TO_UDINT(BlobResults[i + 1].CenterOfMass[1]) + 20,
							 TCVN_FT_HERSHEY_DUPLEX,
							 2,
							 GVL_VisionColor.ColorMagenta,
							 hr);
	END_FOR
END_IF

// Place the Block ID in White and in Black text in the upper left corner of the image
Image_ID_NumText := ULINT_TO_STRING(ImageCount);
hr				 := F_VN_PutTextExp(Image_ID_NumText,
									ipImageIn,
									nX,
									nY,
									TCVN_FT_HERSHEY_SIMPLEX,
									1.5,
									GVL_VisionColor.ColorWhite,
									3,
									TCVN_LT_8_CONNECTED,
									FALSE,
									hr);

hr := F_VN_PutTextExp(Image_ID_NumText,
					  ipImageIn,
					  nX,
					  nY + 50,
					  TCVN_FT_HERSHEY_SIMPLEX,
					  1.5,
					  GVL_VisionColor.ColorBlack,
					  3,
					  TCVN_LT_8_CONNECTED,
					  FALSE,
					  hr);

// Place the Block ID in White and in Black text in the upper left corner of the image
hr := F_VN_PutTextExp(Image_ID_NumText,
					  ipImageRes,
					  nX,
					  nY,
					  TCVN_FT_HERSHEY_SIMPLEX,
					  1.5,
					  GVL_VisionColor.ColorWhite,
					  3,
					  TCVN_LT_8_CONNECTED,
					  FALSE,
					  hr);

hr := F_VN_PutTextExp(Image_ID_NumText,
					  ipImageRes,
					  nX,
					  nY + 50,
					  TCVN_FT_HERSHEY_SIMPLEX,
					  1.5,
					  GVL_VisionColor.ColorBlack,
					  3,
					  TCVN_LT_8_CONNECTED,
					  FALSE,
					  hr);

// Display Input Image
hr := F_VN_TransformIntoDisplayableImage(ipImageIn, ipImageInDisp, hr);

// Display Result Image
hr := F_VN_TransformIntoDisplayableImage(ipImageRes, ipImageResDisp, hr);

// Display Threshold Image
hr := F_VN_TransformIntoDisplayableImage(ipImageWork, ipImageThresholdDisp, hr);
END_METHOD

METHOD PROTECTED Initialize : BOOL
VAR_INPUT
END_VAR
// Set Parameters

// --------------------------------------------------------------

// - Set fMaxArea to 100000 detect all circles or set it to 10000

// to detect only the small circles
BlobParameters.bFilterByArea		:= TRUE;
BlobParameters.fMinArea				:= 100;
BlobParameters.fMaxArea				:= 100000;
BlobParameters.bFilterByCircularity := TRUE;
BlobParameters.fMinCircularity		:= 0.80;
BlobParameters.fMinThreshold		:= 70;
BlobParameters.fThresholdStep		:= 0;

_LightBackground := TRUE;

Initialize := TRUE;
END_METHOD

END_FUNCTION_BLOCK

// Vision/VisionTask/FB_VisionCameraBase
FUNCTION_BLOCK ABSTRACT FB_VisionCameraBase EXTENDS FB_ComponentBase IMPLEMENTS I_CameraBase
VAR
	// Vision Related
	hr		   : HRESULT;
	Camera	   : FB_VN_SimpleCameraControl;
	ipImageIn  : ITcVnImage;
	ImageCount : ULINT;

	//Inputs to Camera
	RunVision		AT %I* : BOOL;
	SoftwareTrigger AT %I* : BOOL;
	Reset			AT %I* : BOOL;

	//Outputs From Camera (Property)
	CameraState		 AT %Q* : ETcVnCameraState;
	ResultsAvailable AT %Q* : BOOL;
	NumberOfResults	 AT %Q* : UDINT;
	Results			 AT %Q* : ARRAY[1..Parameters_Vision.MAX_RESULTS_BUFFER_BYTES] OF BYTE;
	VisionError		 AT %Q* : BOOL;
	VisionErrorID	 AT %Q* : UDINT;

	//Read Write Data
	_ReadData		: BOOL;
	_ReadAddress	: UDINT;
	_WriteData		: BOOL;
	_WriteValue		: UDINT;
	_WriteAddress	: UDINT;
	_ReadDataResult : BOOL;
	_ReadDataValue	: UDINT;
	_ReadDataValid	: BOOL;
	_WriteDataDone	: BOOL;

	//Camera Addresses
	_ExposureAddress : UDINT; //Default is zero and checked when asked to write
	_GainAddress	 : UDINT;

	//Camera Parameter Read/Write Section ******************************************************************
	WriteCamera			  : FB_VN_WriteRegister_UDINT;
	ReadCamera			  : FB_VN_ReadRegister_UDINT;
	ReadValue			  : UDINT;
	ReadCamera_FTRIG	  : F_TRIG;
	ReadCameraError_RTRIG : R_TRIG;

	// Timing Statistics
	SysTimeAtImageArrive : ULINT; // system time units = 1 nS
	SysTimeAtTrigger	 : ULINT; // system time units = 1 nS
	SysTimeAfterProcess	 : ULINT; // system time units = 1 nS
	_ProcessTime		 : LREAL;
	_TriggerToImageTime	 : LREAL;
	_TotalTime			 : LREAL;

	//Read/Write params
	tmpCamParamRead		  : ST_CameraReadWrite;
	tmpCamReadData		  : ST_CameraReadWrite;
	ReadCameraData_RTRIG  : R_TRIG;
	WriteCameraData_RTRIG : R_TRIG;

	//Trigger support
	SoftwareTrigger_RTRIG : R_TRIG;
	HMI_Trigger			  : BOOL;

	//HMI
	VisionBase_HMI : ST_VisionBase_HMI;

	//Generic Results
	FeedbackResults : ARRAY[1..100] OF ST_VisionResults;

	// Image Infos
	PixelFormat : TcVnPixelFormat;

	//HRESULT
	hrFunc : HRESULT;

	// Image Interfaces	
	ipImageInDisp		 : ITcVnDisplayableImage;
	ipImageRes			 : ITcVnImage;
	ipImageResDisp		 : ITcVnDisplayableImage;
	ipImageWork			 : ITcVnImage;
	ipImageThresholdDisp : ITcVnDisplayableImage;

	//Properties
	_LightBackground : BOOL;

	// Parameters for Blob
	BlobParameters : TcVnParamsBlobDetection;

	// Watchdog
	hrWD	  : HRESULT;
	tStop	  : DINT := 5000;
	tRest	  : DINT;
	nFraction : UDINT;

	// Sample Specific Variables
	ipContourList : ITcVnContainer;
END_VAR

PROPERTY LightBackground : BOOL
GET
LightBackground := _LightBackground;
END_GET
SET
_LightBackground := LightBackground;
END_SET
END_PROPERTY

PROPERTY ExposureAddress : UDINT
SET
_ExposureAddress := ExposureAddress;
END_SET
END_PROPERTY

PROPERTY GainAddress : UDINT
SET
_GainAddress := GainAddress;
END_SET
END_PROPERTY

METHOD PUBLIC CyclicLogic
SUPER^.CyclicLogic();

// Do the camera logic
CameraState := Camera.GetState();
CASE CameraState OF
	// Initializing States to get to opened
	TCVN_CS_INITIAL, TCVN_CS_INITIALIZING, TCVN_CS_INITIALIZED, TCVN_CS_OPENING:
		hr := Camera.StartAcquisition();
		IF CameraState = TCVN_CS_INITIALIZED THEN
			VisionError := FALSE;
		END_IF

	// In opened, continue if application asks to run
	TCVN_CS_OPENED:
		IF RunVision THEN
			hr := Camera.StartAcquisition();
		END_IF

	// Always call another StartAquisition when in that state
	TCVN_CS_STARTACQUISITION:
		hr := Camera.StartAcquisition();

	// Response to the Triggering is to TriggerImage again
	TCVN_CS_TRIGGERING:
		hr := Camera.TriggerImage();

	// Waiting for image or application asked to stop running
	TCVN_CS_ACQUIRING:
		hr := Camera.GetCurrentImage(ipImageIn);

		// Check if new Image was received
		IF SUCCEEDED(hr) AND ipImageIn <> 0 THEN
			SysTimeAtImageArrive := F_GetActualDcTime64(); // get system time at new image
			ImageCount			 := ImageCount + 1;
			ProcessImage();
			SysTimeAfterProcess := F_GetActualDcTime64();
			ResultsAvailable	:= TRUE;
			_ProcessTime		:= TO_LREAL(SysTimeAfterProcess - SysTimeAtImageArrive) / TO_LREAL(Tc2_EtherCAT.EC_DCTIME_TICKSPERMSEC64);
			_TriggerToImageTime := TO_LREAL(SysTimeAtImageArrive - SysTimeAtTrigger) / TO_LREAL(Tc2_EtherCAT.EC_DCTIME_TICKSPERMSEC64);
			_TotalTime			:= TO_LREAL(SysTimeAfterProcess - SysTimeAtTrigger) / TO_LREAL(Tc2_EtherCAT.EC_DCTIME_TICKSPERMSEC64);
		ELSIF NOT RunVision THEN
			Camera.StopAcquisition();
		END_IF

	// Stop acqusition requires another call to StopAcquisiton
	TCVN_CS_STOPACQUISITION:
		hr := Camera.StopAcquisition();

	///UH oh.  We are in an error state  try to reset and initialize
	TCVN_CS_ERROR:
		VisionError			:= TRUE;
		hr := Camera.Reset();
END_CASE

//Handle Triggering here
SoftwareTrigger_RTRIG(CLK := (SoftwareTrigger OR HMI_Trigger));
IF SoftwareTrigger_RTRIG.Q THEN
	ResultsAvailable := FALSE;
	hr				 := Camera.TriggerImage();
	IF SUCCEEDED(hr) THEN
		SysTimeAtTrigger := F_GetActualDcTime64();
	END_IF
END_IF

(* Read/Write Camera Data ****************************************************************************
 Check for data in Process Image*)
ReadCameraData_RTRIG(CLK := _ReadData);
IF ReadCameraData_RTRIG.Q THEN
	_ReadDataResult		:= FALSE;
	ReadCamera.nAddress := _ReadAddress;
	ReadCamera.bRead	:= TRUE;
END_IF

ReadCamera(nEndian := 0, nTimeout := T#5S);
ReadCameraError_RTRIG(Clk := ReadCamera.bError AND ReadCamera.bRead AND NOT ReadCamera.bBusy);
ReadCamera.bRead := FALSE;
ReadCamera_FTRIG(CLK := ReadCamera.bBusy);
IF ReadCamera_FTRIG.Q OR ReadCameraError_RTRIG.Q THEN
	IF ReadCamera.bError THEN //ADSERR_DEVICE_BUSY
		_ReadDataResult := TRUE;
		_ReadDataValid	:= FALSE;
	ELSE
		_ReadDataResult := TRUE;
		_ReadDataValue	:= ReadCamera.nValue;
		_ReadDataValid	:= TRUE;
	END_IF
END_IF

WriteCameraData_RTRIG(CLK := _WriteData);

// Check Queue of parameters and Write to Camera
IF WriteCameraData_RTRIG.Q THEN
	_WriteDataDone		 := FALSE;
	WriteCamera.nAddress := _WriteAddress;
	WriteCamera.nValue	 := _WriteValue;
	WriteCamera.bWrite	 := TRUE;
END_IF

WriteCamera(nEndian := 0, nTimeout := T#5S);
WriteCamera.bWrite := FALSE;
IF _WriteData AND (NOT WriteCamera.bBusy OR WriteCamera.bError) THEN
	_WriteDataDone := TRUE;
END_IF

HMICommunication();
END_METHOD

METHOD PROTECTED HMICommunication
VAR_INPUT
END_VAR

VAR_INST
	Trigger_RTRIG	   : R_TRIG;
	ReadExposure_RTRIG : R_TRIG;
	ReadGain_RTRIG	   : R_TRIG;
	SetExposure_RTRIG  : R_TRIG;
	SetGain_RTRIG	   : R_TRIG;
	ReadGain		   : BOOL;
	ReadExposure	   : BOOL;
	SetGain			   : BOOL;
	SetExposure		   : BOOL;
END_VAR
Trigger_RTRIG(CLK := VisionBase_HMI.Command.Trigger);
ReadExposure_RTRIG(CLK := VisionBase_HMI.Config.ReadExposure);
ReadGain_RTRIG(CLK := VisionBase_HMI.Config.ReadGain);
SetExposure_RTRIG(CLK := VisionBase_HMI.Config.SetExposure);
SetGain_RTRIG(CLK := VisionBase_HMI.Config.SetGain);

// handle the request to run vision
IF ComponentBase_HMI.Status.HMIControlAvailable THEN
	IF VisionBase_HMI.Command.StartAquisition THEN
		RunVision := TRUE;
	ELSIF VisionBase_HMI.Command.StopAquisition THEN
		RunVision := FALSE;
	END_IF

	IF ReadExposure_RTRIG.Q AND NOT _ReadData THEN
		ReadExposure := TRUE;
		_ReadAddress := _ExposureAddress;
		_ReadData	 := TRUE;
	ELSIF _ReadDataResult AND ReadExposure THEN
		_ReadData								:= FALSE;
		_ReadDataResult							:= FALSE;
		ReadExposure							:= FALSE;
		VisionBase_HMI.Config.ReadExposureValue := _ReadDataValue;
	END_IF

	IF ReadGain_RTRIG.Q AND NOT _ReadData THEN
		ReadGain	 := TRUE;
		_ReadAddress := _GainAddress;
		_ReadData	 := TRUE;
	ELSIF _ReadDataResult AND ReadGain THEN
		_ReadData							:= FALSE;
		_ReadDataResult						:= FALSE;
		ReadGain							:= FALSE;
		VisionBase_HMI.Config.ReadGainValue := _ReadDataValue;
	END_IF

	IF SetExposure_RTRIG.Q AND NOT _WriteData THEN
		_WriteData	  := TRUE;
		SetExposure	  := TRUE;
		_WriteAddress := _ExposureAddress;
		_WriteValue	  := VisionBase_HMI.Config.Exposure;
	ELSIF _WriteDataDone AND SetExposure THEN
		SetExposure	   := FALSE;
		_WriteDataDone := FALSE;
		_WriteData	   := FALSE;
	END_IF

	IF SetGain_RTRIG.Q AND NOT _WriteData THEN
		SetGain		  := TRUE;
		_WriteData	  := TRUE;
		_WriteAddress := _GainAddress;
		_WriteValue	  := VisionBase_HMI.Config.Gain;
	ELSIF _WriteDataDone AND SetGain THEN
		SetGain		   := FALSE;
		_WriteDataDone := FALSE;
		_WriteData	   := FALSE;
	END_IF

	HMI_Trigger := Trigger_RTRIG.Q;
ELSE
	_ReadData		:= FALSE;
	_ReadDataResult := FALSE;
END_IF

VisionBase_HMI.Status.VisionRunning := RunVision;
VisionBase_HMI.Status.CameraState	:= CameraState;
VisionBase_HMI.Status.ElementsFound := NumberOfResults;
END_METHOD

METHOD PUBLIC  ProcessImage
// Convert Images into the necessary color space
hr := F_VN_GetPixelFormat(ipImageIn, PixelFormat, hr);
IF PixelFormat.nChannels = 3 THEN
	hr := F_VN_CopyImage(ipImageIn, ipImageRes, hr);
	hr := F_VN_ConvertColorSpace(ipImageRes,
								 ipImageIn,
								 TCVN_CST_RGB_TO_GRAY,
								 hr);
ELSE
	hr := F_VN_ConvertColorSpace(ipImageIn,
								 ipImageRes,
								 TCVN_CST_Gray_TO_RGB,
								 hr);
END_IF

// Image Segementation
IF _LightBackground THEN
	hr := F_VN_Threshold(ipImageIn,
						 ipImageWork,
						 BlobParameters.fMinThreshold,
						 255,
						 eThresholdType := TCVN_TT_BINARY_INV,
						 hr);
ELSE
	hr := F_VN_Threshold(ipImageIn,
						 ipImageWork,
						 BlobParameters.fMinThreshold,
						 255,
						 eThresholdType := TCVN_TT_BINARY,
						 hr);
END_IF

// Start Watchdog - DetectBlobs - Stop Watchdog
hrWD   := F_VN_StartRelWatchdog(tStop, S_OK);
hrFunc := F_VN_DetectBlobs(ipSrcImage	  := ipImageWork,
						   ipBlobContours := ipContourList,
						   stParams		  := BlobParameters,
						   hrPrev		  := hr);

hrWD := F_VN_StopWatchdog(hrWD, tRest => tRest, nFractionProcessed => nFraction);
END_METHOD

METHOD ReadParamUDINT : BOOL
VAR_INPUT
	Address : UDINT;
END_VAR

VAR_IN_OUT
	Value : UDINT;
	Valid : BOOL;
END_VAR
ReadParamUDINT := FALSE;
IF NOT _ReadData THEN
	_ReadData := TRUE;
ELSIF _ReadDataResult THEN
	_ReadData		:= FALSE;
	_ReadDataResult := FALSE;
	Valid			:= _ReadDataValid;
	Value			:= _ReadDataValue;
	ReadParamUDINT	:= TRUE;
END_IF
END_METHOD

METHOD SetParamUDINT : BOOL
VAR_INPUT
	Value	: UDINT;
	Address : UDINT;
END_VAR
SetParamUDINT := FALSE;
IF NOT _WriteData THEN
	_WriteData := TRUE;
	_WriteAddress := Address;
	_WriteValue := Value;
ELSIF _WriteDataDone THEN
	_WriteDataDone := FALSE;
	_WriteData := FALSE;
	SetParamUDINT := TRUE;
END_IF
END_METHOD

END_FUNCTION_BLOCK

// Vision/VisionTask/I_CameraBase
INTERFACE I_CameraBase

METHOD CyclicLogic
VAR_INPUT
END_VAR
END_METHOD

METHOD ProcessImage
VAR_INPUT
END_VAR
END_METHOD

END_INTERFACE

// Vision/VisionTask/FB_CameraParameterBuffer
FUNCTION_BLOCK FB_CameraParameterBuffer
VAR
	buffer : FB_MemRingBuffer;
	bufferData : ARRAY[0..100] OF UDINT;
END_VAR

METHOD AddData : BOOL
VAR_INPUT
	data : ST_CameraReadWrite;
END_VAR
buffer(pWrite:=ADR(data),cbWrite:=SIZEOF(data));

buffer.A_AddTail();
END_METHOD

PROPERTY BufferCount : UDINT
GET
BufferCount := buffer.nCount;
END_GET
END_PROPERTY

METHOD GetData
VAR_OUTPUT
	data : ST_CameraReadWrite;
END_VAR
buffer(pRead := ADR(data), cbRead := SIZEOF(data));
buffer.A_GetHead();
END_METHOD

METHOD ReadData : BOOL
VAR_OUTPUT
	data : ST_CameraReadWrite;
END_VAR
buffer(pRead := ADR(data), cbRead := SIZEOF(data));
buffer.A_GetHead();
buffer.A_RemoveHead();
END_METHOD

METHOD ResetData : BOOL
VAR_INPUT
END_VAR
buffer(pBuffer:=ADR(bufferData),cbBuffer:=SIZEOF(bufferData));
buffer.A_Reset();
END_METHOD

END_FUNCTION_BLOCK

// Vision/VisionTask/FB_VideoPlaybackControl
FUNCTION_BLOCK FB_VideoPlaybackControl EXTENDS FB_ListenerBase2 IMPLEMENTS I_CyclicFB
VAR
	//Base FB
	_Busy	 : BOOL := TRUE;
	_Error	 : BOOL;
	_ErrorID : UDINT;

	//Cyclic FB
	_InitComplete : BOOL;

	// Video Playback Control
	_CameraID : UINT;

	//EnableImagesToBuffer : BOOL;
	TriggerVideoCapture : BOOL;
	VideoCaptureState	: INT;

	// Ring Buffer information
	BufferImageRing : ARRAY[1..Parameters_Vision.MAX_NUMBER_IMAGES_2_VIDEO] OF ITcVnImage;
	BufferIndex		: INT := 1;

	//BufferImageSaveIndex	  : UINT;
	WriteImageWaitResult	  : BOOL;
	ipImageForVideoRingBuffer : ITcVnImage;
	ipImageToSave			  : ITcVnImage;
	WriteFileState			  : INT;
	sImageToSaveName		  : STRING;
	fbWriteImage			  : FB_VN_WriteImage;
	SysTimeAtFileWrite		  : ULINT;
	_fbEvent				  : FB_TcEvent;
	sFileName1				  : T_MaxString;

	//Properties
	_ImageReductionFactor : LREAL := 1; // This is the amount of reduction to image for making video Default := 1;
	_ImageSourceDirectory : STRING;
	_VideoOutputDirectory : STRING;
	_FramesPerSecond	  : UINT;

	//Alarm data
	sJsonAttribute	 : STRING(10000);
	JSONFilter		 : FB_TcEventFilter;
	JSONString		 : T_MaxString := '{"CreateVideo": 1}';
	_Subscribe		 : BOOL		   := TRUE;
	_Unsubscribe	 : BOOL;
	_Subscribed		 : BOOL;
	MissedEventCount : UDINT;

	//Image count value
	ImageWriteCount : UINT;

	//Delay after alarm to wait then do work
	AlarmDelay		: TON;
	_AlarmDelayTime : TIME;
	StopImageAdding : BOOL;
END_VAR

PROPERTY Busy : BOOL
GET
Busy := _Busy;
END_GET
END_PROPERTY

PROPERTY Error : BOOL
GET
Error := _Error;
END_GET
END_PROPERTY

PROPERTY ErrorID : UDINT
GET
ErrorID := _ErrorID;
END_GET
END_PROPERTY

METHOD CyclicLogic
VAR
	hr				: HRESULT;
	tmpIndex		: INT;
	systemTimeNow	: TIMESTRUCT;
	tmpString		: STRING;
	EventTimestamp1 : TimeStruct;
	sDump			: STRING;
END_VAR

VAR_INST
	x : INT;
END_VAR
IF NOT _InitComplete THEN
	_InitComplete := TRUE;
END_IF

// Call the Listener Execute
Execute();
IF _Subscribe THEN
	_Subscribe := FALSE;
	JSONFilter.Clear().JsonAttribute.Value.EqualTo(JSONString); //define all events (messages and alarms) from this eventclass   
	hr := Subscribe2(JSONFilter);								//subscribe to retrieve defined events
	IF SUCCEEDED(hr) THEN
		_Subscribed := TRUE;
	END_IF
END_IF

IF _Unsubscribe THEN
	_Unsubscribe := FALSE;
	hr			 := Unsubscribe();
	IF SUCCEEDED(hr) THEN
		_Subscribed := FALSE;
	END_IF
END_IF

CASE VideoCaptureState OF
	0:
		IF TriggerVideoCapture THEN
			x				  := 1;
			VideoCaptureState := 10;
		END_IF

	10:
		IF AlarmDelay.Q THEN
			StopImageAdding := TRUE;
			VideoCaptureState := 15;
		END_IF
	
	15:	
		tmpIndex := BufferIndex + x - 1;
		IF tmpIndex > TO_INT(Parameters_Vision.MAX_NUMBER_IMAGES_2_VIDEO) THEN
			tmpIndex := tmpIndex - TO_INT(Parameters_Vision.MAX_NUMBER_IMAGES_2_VIDEO);
		END_IF

		IF WriteImage(Index := x, BufferImageSaveNameIndex := TmpIndex) THEN
			x := x + 1;
		END_IF

		IF x > TO_INT(Parameters_Vision.MAX_NUMBER_IMAGES_2_VIDEO) THEN
			TriggerVideoCapture := FALSE;
			StopImageAdding := FALSE;
			VideoCaptureState	:= 20;
		END_IF

	20:
		EventTimestamp1 := FILETIME64_TO_SYSTEMTIME(_fbevent.nTimestamp);
		sFileName1		:= SYSTEMTIME_TO_STRING(EventTimestamp1);
		FindAndReplaceChar(ADR(sFileName1),
						   ':',
						   '-',
						   ADR(sFileName1),
						   SIZEOF(sFileName1));

		FindAndSplitChar(sSeparatorChar	  := '.',
						 pSrcString		  := ADR(sFileName1),
						 pLeftString	  := ADR(sFileName1),
						 nLeftSize		  := SIZEOF(sFileName1),
						 pRightString	  := ADR(sDump),
						 nRightSize		  := SIZEOF(sDump),
						 bSearchFromRight := FALSE);

		sFileName1											:= CONCAT(sFileName1, '.avi');
		GVL_Image2Video.CameraData[_CameraID].VideoFilename := sFileName1;
		GVL_Image2Video.CameraData[_CameraID].VideoCreate	:= TRUE;
		VideoCaptureState									:= 30;

	30:
		IF GVL_Image2Video.CameraData[_CameraID].VideoCreated THEN
			GVL_Image2Video.CameraData[_CameraID].VideoCreate  := FALSE;
			GVL_Image2Video.CameraData[_CameraID].VideoCreated := FALSE;
			VideoCaptureState								   := 0;
		END_IF
END_CASE

IF GVL_Image2Video.CameraData[_CameraID].Heartbeat THEN
	GVL_Image2Video.CameraData[_CameraID].Heartbeat := FALSE;
END_IF

AlarmDelay(IN:= VideoCaptureState =10, PT:=_AlarmDelayTime);

GVL_Image2Video.CameraData[_CameraID].VideoPathSource := _VideoOutputDirectory;
GVL_Image2Video.CameraData[_CameraID].ImagePathSource := _ImageSourceDirectory;
GVL_Image2Video.CameraData[_CameraID].VideoFPS		  := _FramesPerSecond;
END_METHOD

PROPERTY InitComplete : BOOL
GET
InitComplete := _InitComplete;
END_GET
END_PROPERTY

METHOD Execute : HRESULT
VAR_INPUT
END_VAR
Execute := SUPER^.Execute();
END_METHOD

METHOD OnAlarmRaised : HRESULT
VAR_INPUT
	fbEvent : REFERENCE TO FB_TcEvent;
END_VAR

VAR 
	hr : HRESULT;
END_VAR
// This is where we actually do the work
IF NOT TriggerVideoCapture THEN
	TriggerVideoCapture := TRUE;
	ImageWriteCount := 1;
	hr					:= fbEvent.GetJsonAttribute(sJsonAttribute, SIZEOF(sJsonAttribute));
	_fbEvent:=fbevent;
ELSE
	MissedEventCount := MissedEventCount + 1;
END_IF

OnAlarmRaised := S_OK;
END_METHOD

PROPERTY SubscribedEvents : BOOL
GET
SubscribedEvents := _Subscribed;
END_GET
END_PROPERTY

PROPERTY SubscribeEvents : BOOL
SET
_Subscribe := SubscribeEvents;
END_SET
END_PROPERTY

PROPERTY UnsubscribeEvents : BOOL
SET
_Unsubscribe := UnsubscribeEvents;
END_SET
END_PROPERTY

METHOD AddImage : BOOL
VAR_INPUT
	ipImageIn : ITcVnImage; // Image to be added to buffer
END_VAR

VAR
	hr						  : HRESULT;
	hrWD1					  : HRESULT;
	tStop1					  : DINT := 20000;
	tRest1					  : DINT;
	ImageInfo				  : TcVnImageInfo;
	ImagePixelFormatChannels  : BYTE;
	ImageEffectivePixelSize	  : UINT;
	ImageInWidth			  : UDINT;
	ImageInHeight			  : UDINT;
	ImageSmallWidth			  : UDINT;
	ImageSmallHeight		  : UDINT;
END_VAR
IF NOT StopImageAdding THEN
	hr						 := F_VN_GetImageInfo(ipImage := ipImageIn, stImageInfo := ImageInfo, hrPrev := S_OK);
	ImagePixelFormatChannels := ImageInfo.stPixelFormat.nChannels;
	ImageEffectivePixelSize	 := ImageInfo.stPixelFormat.nElementSize;
	ImageInWidth			 := ImageInfo.nWidth;
	ImageInHeight			 := ImageInfo.nHeight;
	IF _ImageReductionFactor <> 1 THEN
		ImageSmallWidth	 := LREAL_TO_UDINT(UDINT_TO_LREAL(ImageInWidth) * _ImageReductionFactor);
		ImageSmallHeight := LREAL_TO_UDINT(UDINT_TO_LREAL(ImageInHeight) * _ImageReductionFactor);

		// Image Width and Height must be even for video conversion
		IF (ImageSmallWidth MOD 2) <> 0 THEN // Check if "Odd"
			ImageSmallWidth := ImageSmallWidth - 1;
		END_IF

		IF (ImageSmallHeight MOD 2) <> 0 THEN // Check if "Odd"
			ImageSmallHeight := ImageSmallHeight - 1;
		END_IF

